C01831=1180.589,-28.436,-43.690,179.742,5.773,149.102
C01832=1180.584,-28.186,-43.703,179.744,5.773,149.101
C01833=1180.579,-27.936,-43.716,179.746,5.773,149.101
C01834=1180.573,-27.686,-43.728,179.749,5.774,149.100
C01835=1180.568,-27.437,-43.740,179.751,5.774,149.100
C01836=1180.563,-27.188,-43.753,179.753,5.775,149.099
C01837=1180.557,-26.938,-43.766,179.756,5.775,149.098
C01838=1180.553,-26.687,-43.778,179.758,5.776,149.098
C01839=1180.547,-26.438,-43.791,179.761,5.777,149.097
C01840=1180.542,-26.189,-43.803,179.763,5.776,149.096
C01841=1180.537,-25.939,-43.816,179.766,5.777,149.096
C01842=1180.532,-25.689,-43.828,179.768,5.777,149.095
C01843=1180.527,-25.439,-43.841,179.770,5.778,149.094
C01844=1180.522,-25.190,-43.854,179.773,5.778,149.094
C01845=1180.517,-24.941,-43.866,179.775,5.779,149.093
C01846=1180.512,-24.691,-43.878,179.778,5.780,149.093
C01847=1180.506,-24.442,-43.891,179.780,5.779,149.092
C01848=1180.501,-24.191,-43.904,179.782,5.780,149.091
C01849=1180.496,-23.922,-43.917,179.785,5.781,149.091
C01850=1180.491,-23.652,-43.931,179.787,5.781,149.090
C01851=1180.485,-23.382,-43.945,179.790,5.781,149.089
C01852=1180.479,-23.113,-43.958,179.793,5.782,149.089
C01853=1180.474,-22.863,-43.971,179.795,5.782,149.088
C01854=1180.469,-22.613,-43.984,179.798,5.783,149.087
C01855=1180.463,-22.364,-43.997,179.800,5.784,149.087
C01856=1180.458,-22.115,-44.009,179.803,5.784,149.086
C01857=1180.453,-21.865,-44.022,179.806,5.785,149.085
C01858=1180.449,-21.615,-44.035,179.808,5.785,149.085
C01859=1180.443,-21.365,-44.047,179.810,5.785,149.084
C01860=1180.437,-21.116,-44.060,179.813,5.785,149.084
C01861=1180.433,-20.866,-44.073,179.815,5.786,149.083
C01862=1180.428,-20.616,-44.086,179.817,5.787,149.082
C01863=1180.423,-20.367,-44.098,179.820,5.787,149.082
C01864=1180.417,-20.118,-44.111,179.822,5.788,149.081
C01865=1180.412,-19.867,-44.124,179.825,5.788,149.080
C01866=1180.407,-19.618,-44.137,179.828,5.789,149.080
C01867=1180.402,-19.369,-44.150,179.830,5.789,149.079
C01868=1180.397,-19.119,-44.162,179.832,5.789,149.079
C01869=1180.392,-18.869,-44.176,179.834,5.790,149.078
C01870=1180.386,-18.620,-44.188,179.837,5.790,149.077
C01871=1180.381,-18.370,-44.201,179.839,5.791,149.077
C01872=1180.377,-18.120,-44.214,179.842,5.792,149.076
C01873=1180.371,-17.871,-44.227,179.845,5.792,149.075
C01874=1180.366,-17.621,-44.240,179.847,5.793,149.075
C01875=1180.361,-17.371,-44.253,179.849,5.793,149.074
C01876=1180.355,-17.122,-44.266,179.852,5.794,149.074
C01877=1180.350,-16.872,-44.278,179.854,5.794,149.073
C01878=1180.346,-16.622,-44.291,179.856,5.794,149.072
C01879=1180.341,-16.373,-44.304,179.859,5.795,149.072
C01880=1180.335,-16.124,-44.317,179.862,5.795,149.071
C01881=1180.330,-15.873,-44.330,179.864,5.796,149.071
C01882=1180.325,-15.624,-44.343,179.866,5.796,149.070
C01883=1180.319,-15.375,-44.356,179.869,5.797,149.069
C01884=1180.315,-15.125,-44.369,179.871,5.798,149.069
C01885=1180.310,-14.875,-44.382,179.874,5.798,149.068
C01886=1180.304,-14.626,-44.395,179.877,5.799,149.067
C01887=1180.300,-14.376,-44.408,179.878,5.799,149.067
C01888=1180.294,-14.127,-44.421,179.881,5.799,149.066
C01889=1180.289,-13.877,-44.434,179.884,5.800,149.065
C01890=1180.284,-13.627,-44.447,179.886,5.800,149.065
C01891=1180.278,-13.378,-44.460,179.888,5.801,149.064
C01892=1180.273,-13.128,-44.473,179.891,5.801,149.064
C01893=1180.269,-12.878,-44.486,179.894,5.802,149.063
C01894=1180.263,-12.629,-44.500,179.896,5.803,149.062
C01895=1180.258,-12.379,-44.513,179.899,5.803,149.062
C01896=1180.253,-12.130,-44.525,179.901,5.804,149.061
C01897=1180.247,-11.880,-44.539,179.903,5.804,149.061
C01898=1180.243,-11.630,-44.552,179.906,5.805,149.060
C01899=1180.237,-11.381,-44.566,179.909,5.805,149.059
C01900=1180.233,-11.131,-44.579,179.910,5.805,149.059
C01901=1180.227,-10.882,-44.592,179.913,5.806,149.058
C01902=1180.222,-10.632,-44.605,179.916,5.806,149.057
C01903=1180.218,-10.383,-44.618,179.918,5.807,149.057
C01904=1180.212,-10.133,-44.631,179.920,5.808,149.056
C01905=1180.207,-9.883,-44.644,179.923,5.808,149.055
C01906=1180.201,-9.634,-44.657,179.926,5.809,149.055
C01907=1180.197,-9.384,-44.671,179.928,5.809,149.054
C01908=1180.191,-9.135,-44.684,179.931,5.810,149.054
C01909=1180.187,-8.885,-44.697,179.933,5.810,149.053
C01910=1180.181,-8.635,-44.710,179.935,5.811,149.052
C01911=1180.177,-8.386,-44.724,179.938,5.812,149.052
C01912=1180.171,-8.136,-44.737,179.941,5.812,149.051
C01913=1180.166,-7.887,-44.750,179.943,5.813,149.050
C01914=1180.161,-7.637,-44.764,179.945,5.813,149.050
C01915=1180.156,-7.388,-44.777,179.948,5.814,149.049
C01916=1180.150,-7.137,-44.790,179.950,5.813,149.049
C01917=1180.146,-6.889,-44.804,179.952,5.814,149.048
C01918=1180.140,-6.638,-44.817,179.955,5.815,149.047
C01919=1180.136,-6.390,-44.830,179.958,5.815,149.047
C01920=1180.130,-6.139,-44.844,179.960,5.816,149.046
C01921=1180.125,-5.890,-44.857,179.963,5.817,149.046
C01922=1180.120,-5.640,-44.871,179.965,5.817,149.045
C01923=1180.115,-5.391,-44.884,179.967,5.818,149.044
C01924=1180.110,-5.141,-44.898,179.970,5.818,149.044
C01925=1180.105,-4.892,-44.910,179.973,5.819,149.043
C01926=1180.100,-4.641,-44.924,179.975,5.819,149.042
C01927=1180.094,-4.392,-44.938,179.977,5.820,149.042
C01928=1180.090,-4.142,-44.951,179.980,5.821,149.041
C01929=1180.084,-3.893,-44.965,179.983,5.821,149.040
C01930=1180.080,-3.643,-44.978,179.985,5.822,149.040
C01931=1180.074,-3.394,-44.992,179.988,5.822,149.039
C01932=1180.069,-3.144,-45.005,179.990,5.823,149.039
C01933=1180.064,-2.895,-45.019,179.992,5.824,149.038
C01934=1180.059,-2.645,-45.032,179.995,5.824,149.037
C01935=1180.054,-2.396,-45.046,179.998,5.825,149.037
C01936=1180.049,-2.146,-45.059,180.000,5.825,149.036
C01937=1180.044,-1.896,-45.073,-179.997,5.826,149.036
C01938=1180.039,-1.647,-45.086,-179.995,5.826,149.035
C01939=1180.034,-1.397,-45.100,-179.993,5.827,149.035
C01940=1180.028,-1.148,-45.113,-179.990,5.828,149.034
C01941=1180.023,-0.898,-45.127,-179.987,5.828,149.033
C01942=1180.018,-0.649,-45.140,-179.985,5.829,149.032
C01943=1180.013,-0.399,-45.154,-179.982,5.829,149.032
C01944=1180.008,-0.150,-45.168,-179.980,5.830,149.031
C01945=1180.003,0.100,-45.181,-179.977,5.830,149.031
C01946=1179.998,0.350,-45.196,-179.976,5.830,149.030
C01947=1179.993,0.599,-45.208,-179.973,5.831,149.029
C01948=1179.988,0.849,-45.222,-179.970,5.831,149.029
C01949=1179.983,1.099,-45.237,-179.968,5.832,149.028
C01950=1179.977,1.348,-45.249,-179.965,5.833,149.028
C01951=1179.973,1.598,-45.264,-179.963,5.833,149.027
C01952=1179.967,1.847,-45.277,-179.961,5.834,149.026
C01953=1179.961,2.117,-45.292,-179.957,5.835,149.026
C01954=1179.956,2.386,-45.307,-179.955,5.836,149.025
C01955=1179.951,2.655,-45.321,-179.952,5.836,149.024
C01956=1179.945,2.924,-45.336,-179.949,5.837,149.024
C01957=1179.940,3.174,-45.350,-179.947,5.837,149.023
C01958=1179.935,3.423,-45.364,-179.945,5.838,149.023
C01959=1179.929,3.673,-45.378,-179.942,5.838,149.022
C01960=1179.925,3.922,-45.391,-179.939,5.839,149.021
C01961=1179.920,4.172,-45.406,-179.937,5.840,149.021
C01962=1179.915,4.421,-45.419,-179.934,5.840,149.020
C01963=1179.909,4.671,-45.433,-179.932,5.841,149.019
C01964=1179.904,4.921,-45.447,-179.930,5.842,149.019
C01965=1179.900,5.170,-45.461,-179.927,5.842,149.018
C01966=1179.895,5.419,-45.475,-179.924,5.843,149.018
C01967=1179.889,5.670,-45.488,-179.922,5.843,149.017
C01968=1179.884,5.919,-45.502,-179.920,5.844,149.016
C01969=1179.879,6.169,-45.517,-179.917,5.844,149.016
C01970=1179.875,6.418,-45.530,-179.914,5.845,149.015
C01971=1179.869,6.667,-45.544,-179.912,5.846,149.015
C01972=1179.864,6.917,-45.558,-179.909,5.846,149.014
C01973=1179.859,7.167,-45.572,-179.907,5.847,149.013
C01974=1179.853,7.416,-45.586,-179.905,5.847,149.013
C01975=1179.848,7.666,-45.600,-179.902,5.848,149.012
C01976=1179.843,7.915,-45.615,-179.899,5.848,149.011
C01977=1179.839,8.165,-45.628,-179.897,5.849,149.011
C01978=1179.833,8.414,-45.641,-179.894,5.850,149.010
C01979=1179.828,8.664,-45.656,-179.892,5.850,149.010
C01980=1179.823,8.914,-45.670,-179.890,5.851,149.009
C01981=1179.818,9.163,-45.684,-179.887,5.852,149.008
C01982=1179.813,9.413,-45.698,-179.884,5.853,149.008
C01983=1179.808,9.662,-45.712,-179.882,5.854,149.007
C01984=1179.803,9.912,-45.727,-179.879,5.854,149.007
C01985=1179.797,10.161,-45.741,-179.876,5.855,149.006
C01986=1179.793,10.410,-45.754,-179.874,5.855,149.005
C01987=1179.788,10.661,-45.768,-179.871,5.856,149.005
C01988=1179.783,10.910,-45.782,-179.869,5.856,149.004
C01989=1179.777,11.159,-45.796,-179.867,5.857,149.004
C01990=1179.772,11.409,-45.810,-179.864,5.858,149.003
C01991=1179.767,11.659,-45.825,-179.861,5.858,149.002
C01992=1179.763,11.909,-45.839,-179.859,5.859,149.002
C01993=1179.757,12.158,-45.853,-179.857,5.860,149.001
C01994=1179.752,12.407,-45.867,-179.854,5.860,149.000
C01995=1179.747,12.657,-45.881,-179.852,5.861,149.000
C01996=1179.742,12.907,-45.896,-179.849,5.861,148.999
C01997=1179.737,13.156,-45.910,-179.846,5.862,148.999
C01998=1179.732,13.405,-45.924,-179.844,5.863,148.998
C01999=1179.727,13.655,-45.938,-179.842,5.863,148.997
C02000=1179.722,13.905,-45.952,-179.839,5.864,148.997
C02001=1179.717,14.155,-45.967,-179.837,5.865,148.996
C02002=1179.711,14.403,-45.981,-179.834,5.865,148.996
C02003=1179.707,14.653,-45.996,-179.831,5.866,148.995
C02004=1179.702,14.902,-46.010,-179.829,5.867,148.994
C02005=1179.697,15.152,-46.024,-179.826,5.868,148.994
C02006=1179.692,15.402,-46.038,-179.823,5.868,148.993
C02007=1179.687,15.652,-46.053,-179.821,5.869,148.993
C02008=1179.681,15.901,-46.067,-179.819,5.869,148.992
C02009=1179.676,16.150,-46.081,-179.816,5.870,148.991
C02010=1179.671,16.400,-46.095,-179.814,5.871,148.991
C02011=1179.666,16.650,-46.109,-179.811,5.871,148.990
C02012=1179.661,16.899,-46.125,-179.808,5.872,148.989
C02013=1179.656,17.149,-46.139,-179.806,5.873,148.989
C02014=1179.650,17.398,-46.153,-179.804,5.873,148.988
C02015=1179.645,17.648,-46.167,-179.801,5.874,148.988
C02016=1179.640,17.897,-46.182,-179.799,5.874,148.987
C02017=1179.636,18.147,-46.196,-179.796,5.876,148.986
C02018=1179.631,18.396,-46.211,-179.793,5.876,148.986
C02019=1179.626,18.646,-46.225,-179.791,5.877,148.985
C02020=1179.621,18.895,-46.240,-179.788,5.878,148.985
C02021=1179.616,19.145,-46.254,-179.786,5.878,148.984
C02022=1179.610,19.394,-46.269,-179.783,5.879,148.984
C02023=1179.605,19.644,-46.283,-179.781,5.879,148.983
C02024=1179.600,19.893,-46.298,-179.778,5.880,148.982
C02025=1179.595,20.143,-46.312,-179.776,5.881,148.982
C02026=1179.591,20.392,-46.327,-179.773,5.881,148.981
C02027=1179.586,20.642,-46.341,-179.771,5.882,148.980
C02028=1179.580,20.892,-46.356,-179.768,5.883,148.980
C02029=1179.575,21.142,-46.370,-179.765,5.884,148.979
C02030=1179.570,21.391,-46.385,-179.763,5.884,148.979
C02031=1179.565,21.640,-46.400,-179.760,5.885,148.978
C02032=1179.560,21.890,-46.414,-179.758,5.886,148.977
C02033=1179.554,22.139,-46.429,-179.755,5.886,148.977
C02034=1179.549,22.388,-46.443,-179.753,5.887,148.976
C02035=1179.544,22.638,-46.458,-179.750,5.887,148.976
C02036=1179.540,22.887,-46.473,-179.748,5.888,148.975
C02037=1179.535,23.137,-46.487,-179.745,5.889,148.974
C02038=1179.529,23.387,-46.502,-179.742,5.890,148.974
C02039=1179.525,23.636,-46.517,-179.740,5.891,148.973
C02040=1179.520,23.886,-46.531,-179.737,5.891,148.973
C02041=1179.515,24.135,-46.546,-179.735,5.892,148.972
C02042=1179.509,24.385,-46.561,-179.732,5.892,148.971
C02043=1179.504,24.635,-46.575,-179.730,5.893,148.971
C02044=1179.500,24.884,-46.590,-179.727,5.894,148.970
C02045=1179.495,25.133,-46.604,-179.725,5.895,148.970
C02046=1179.489,25.383,-46.620,-179.722,5.896,148.969
C02047=1179.484,25.633,-46.634,-179.719,5.896,148.968
C02048=1179.480,25.882,-46.649,-179.717,5.897,148.968
C02049=1179.474,26.132,-46.664,-179.714,5.898,148.967
C02050=1179.469,26.381,-46.679,-179.712,5.898,148.967
C02051=1179.464,26.630,-46.693,-179.710,5.899,148.966
C02052=1179.459,26.880,-46.709,-179.707,5.900,148.965
C02053=1179.454,27.130,-46.723,-179.704,5.900,148.965
C02054=1179.449,27.379,-46.738,-179.702,5.902,148.964
C02055=1179.444,27.629,-46.753,-179.699,5.902,148.964
C02056=1179.439,27.878,-46.768,-179.696,5.903,148.963
C02057=1179.434,28.147,-46.784,-179.694,5.904,148.962
C02058=1179.428,28.416,-46.800,-179.692,5.904,148.962
C02059=1179.423,28.684,-46.816,-179.688,5.905,148.961
C02060=1179.417,28.954,-46.832,-179.686,5.906,148.960
C02061=1179.412,29.203,-46.847,-179.683,5.906,148.960
C02062=1179.407,29.452,-46.861,-179.681,5.907,148.959
C02063=1179.402,29.702,-46.877,-179.678,5.908,148.959
C02064=1179.397,29.951,-46.891,-179.675,5.909,148.958
C02065=1179.392,30.201,-46.907,-179.673,5.910,148.957
C02066=1179.387,30.450,-46.922,-179.670,5.910,148.957
C02067=1179.382,30.700,-46.936,-179.668,5.911,148.956
C02068=1179.377,30.949,-46.952,-179.665,5.912,148.956
C02069=1179.372,31.198,-46.967,-179.663,5.912,148.955
C02070=1179.366,31.448,-46.982,-179.660,5.914,148.955
C02071=1179.362,31.698,-46.997,-179.657,5.914,148.954
C02072=1179.357,31.947,-47.013,-179.655,5.915,148.953
C02073=1179.352,32.197,-47.027,-179.653,5.916,148.953
C02074=1179.347,32.446,-47.042,-179.650,5.916,148.952
C02075=1179.342,32.696,-47.057,-179.647,5.917,148.951
C02076=1179.337,32.945,-47.072,-179.644,5.918,148.951
C02077=1179.332,33.195,-47.087,-179.642,5.919,148.950
C02078=1179.327,33.444,-47.102,-179.640,5.920,148.950
C02079=1179.321,33.694,-47.117,-179.637,5.920,148.949
C02080=1179.317,33.943,-47.132,-179.634,5.921,148.948
C02081=1179.312,34.193,-47.148,-179.632,5.922,148.948
C02082=1179.307,34.442,-47.163,-179.629,5.923,148.947
C02083=1179.302,34.692,-47.178,-179.626,5.923,148.947
C02084=1179.297,34.941,-47.193,-179.624,5.924,148.946
C02085=1179.291,35.191,-47.209,-179.622,5.925,148.946
C02086=1179.287,35.440,-47.224,-179.619,5.926,148.945
C02087=1179.281,35.689,-47.239,-179.617,5.926,148.944
C02088=1179.277,35.940,-47.254,-179.614,5.928,148.944
C02089=1179.272,36.189,-47.269,-179.611,5.928,148.943
C02090=1179.266,36.438,-47.285,-179.609,5.929,148.943
C02091=1179.262,36.687,-47.300,-179.606,5.929,148.942
C02092=1179.256,36.937,-47.316,-179.604,5.930,148.942
C02093=1179.252,37.186,-47.331,-179.601,5.932,148.941
C02094=1179.247,37.437,-47.346,-179.599,5.932,148.940
C02095=1179.242,37.686,-47.361,-179.596,5.933,148.940
C02096=1179.236,37.935,-47.376,-179.593,5.933,148.939
C02097=1179.231,38.185,-47.392,-179.591,5.934,148.939
C02098=1179.226,38.434,-47.407,-179.588,5.936,148.938
C02099=1179.221,38.683,-47.423,-179.586,5.936,148.937
C02100=1179.217,38.933,-47.438,-179.583,5.937,148.937
C02101=1179.212,39.182,-47.453,-179.580,5.937,148.936
C02102=1179.206,39.432,-47.469,-179.578,5.938,148.936
C02103=1179.202,39.681,-47.484,-179.575,5.940,148.935
C02104=1179.196,39.930,-47.500,-179.572,5.940,148.934
C02105=1179.191,40.181,-47.515,-179.570,5.941,148.934
C02106=1179.186,40.430,-47.530,-179.568,5.942,148.933
C02107=1179.181,40.679,-47.545,-179.565,5.942,148.933
C02108=1179.176,40.929,-47.561,-179.562,5.944,148.932
C02109=1179.172,41.179,-47.576,-179.560,5.944,148.931
C02110=1179.166,41.428,-47.592,-179.557,5.945,148.931
C02111=1179.161,41.677,-47.608,-179.555,5.946,148.930
C02112=1179.156,41.926,-47.623,-179.553,5.946,148.930
C02113=1179.151,42.177,-47.639,-179.549,5.948,148.929
C02114=1179.146,42.426,-47.654,-179.547,5.948,148.929
C02115=1179.142,42.674,-47.670,-179.545,5.949,148.928
C02116=1179.136,42.924,-47.685,-179.542,5.950,148.927
C02117=1179.132,43.174,-47.701,-179.539,5.951,148.927
C02118=1179.126,43.423,-47.717,-179.537,5.952,148.926
C02119=1179.122,43.672,-47.732,-179.534,5.952,148.926
C02120=1179.116,43.922,-47.748,-179.532,5.953,148.925
C02121=1179.111,44.172,-47.764,-179.529,5.954,148.925
C02122=1179.106,44.421,-47.779,-179.526,5.955,148.924
C02123=1179.101,44.670,-47.794,-179.524,5.956,148.923
C02124=1179.097,44.920,-47.810,-179.521,5.956,148.923
C02125=1179.091,45.169,-47.826,-179.519,5.957,148.922
C02126=1179.086,45.419,-47.842,-179.516,5.959,148.922
C02127=1179.082,45.668,-47.857,-179.514,5.959,148.921
C02128=1179.077,45.918,-47.873,-179.511,5.960,148.921
C02129=1179.071,46.167,-47.888,-179.508,5.960,148.920
C02130=1179.066,46.417,-47.904,-179.506,5.962,148.919
C02131=1179.061,46.666,-47.921,-179.503,5.963,148.919
C02132=1179.057,46.915,-47.936,-179.501,5.964,148.918
C02133=1179.052,47.165,-47.952,-179.498,5.964,148.918
C02134=1179.047,47.415,-47.967,-179.495,5.965,148.917
C02135=1179.041,47.664,-47.983,-179.493,5.966,148.917
C02136=1179.037,47.914,-48.000,-179.490,5.967,148.916
C02137=1179.031,48.163,-48.015,-179.488,5.968,148.915
C02138=1179.027,48.412,-48.030,-179.485,5.969,148.915
C02139=1179.022,48.662,-48.046,-179.482,5.969,148.914
C02140=1179.017,48.911,-48.062,-179.480,5.970,148.914
C02141=1179.011,49.160,-48.078,-179.477,5.971,148.913
C02142=1179.007,49.411,-48.094,-179.475,5.973,148.913
C02143=1179.002,49.659,-48.110,-179.472,5.973,148.912
C02144=1178.997,49.909,-48.126,-179.469,5.974,148.911
C02145=1178.991,50.159,-48.142,-179.467,5.974,148.911
C02146=1178.987,50.407,-48.157,-179.464,5.976,148.910
C02147=1178.982,50.657,-48.173,-179.462,5.977,148.910
C02148=1178.977,50.907,-48.189,-179.459,5.977,148.909
C02149=1178.972,51.156,-48.206,-179.457,5.978,148.909
C02150=1178.967,51.406,-48.221,-179.454,5.979,148.908
C02151=1178.962,51.655,-48.237,-179.451,5.980,148.907
C02152=1178.957,51.905,-48.254,-179.449,5.981,148.907
C02153=1178.952,52.154,-48.269,-179.446,5.982,148.906
C02154=1178.947,52.404,-48.285,-179.444,5.983,148.906
C02155=1178.942,52.653,-48.301,-179.441,5.983,148.905
C02156=1178.937,52.903,-48.317,-179.439,5.984,148.905
C02157=1178.932,53.152,-48.334,-179.436,5.986,148.904
C02158=1178.927,53.401,-48.349,-179.433,5.986,148.903
C02159=1178.922,53.651,-48.366,-179.431,5.987,148.903
C02160=1178.917,53.900,-48.381,-179.428,5.988,148.902
C02161=1178.912,54.169,-48.399,-179.425,5.989,148.901
C02162=1178.907,54.437,-48.417,-179.423,5.990,148.901
C02163=1178.901,54.706,-48.434,-179.420,5.991,148.900
C02164=1178.895,54.974,-48.451,-179.417,5.992,148.900
C02165=1178.891,55.224,-48.467,-179.414,5.993,148.899
C02166=1178.886,55.473,-48.483,-179.412,5.994,148.899
C02167=1178.881,55.722,-48.500,-179.409,5.994,148.898
C02168=1178.876,55.972,-48.515,-179.406,5.996,148.897
C02169=1178.871,56.221,-48.532,-179.404,5.996,148.897
C02170=1178.866,56.471,-48.547,-179.401,5.997,148.896
C02171=1178.861,56.720,-48.564,-179.398,5.999,148.896
C02172=1178.856,56.970,-48.580,-179.396,6.000,148.895
C02173=1178.851,57.219,-48.597,-179.393,6.000,148.895
C02174=1178.845,57.469,-48.612,-179.391,6.001,148.894
C02175=1178.841,57.718,-48.629,-179.388,6.002,148.893
C02176=1178.836,57.967,-48.645,-179.385,6.003,148.893
C02177=1178.831,58.217,-48.661,-179.383,6.004,148.892
C02178=1178.826,58.466,-48.678,-179.380,6.005,148.892
C02179=1178.821,58.715,-48.694,-179.378,6.006,148.891
C02180=1178.816,58.965,-48.710,-179.375,6.006,148.891
C02181=1178.812,59.214,-48.727,-179.373,6.008,148.890
C02182=1178.805,59.464,-48.743,-179.370,6.009,148.889
C02183=1178.801,59.713,-48.759,-179.368,6.010,148.889
C02184=1178.796,59.963,-48.776,-179.365,6.011,148.888
C02185=1178.791,60.212,-48.792,-179.362,6.011,148.888
C02186=1178.787,60.462,-48.808,-179.360,6.012,148.887
C02187=1178.782,60.711,-48.825,-179.357,6.014,148.887
C02188=1178.777,60.960,-48.841,-179.354,6.014,148.886
C02189=1178.771,61.210,-48.858,-179.352,6.015,148.886
C02190=1178.766,61.459,-48.874,-179.349,6.017,148.885
C02191=1178.762,61.709,-48.891,-179.346,6.017,148.884
C02192=1178.757,61.958,-48.907,-179.344,6.018,148.884
C02193=1178.752,62.208,-48.923,-179.341,6.019,148.883
C02194=1178.746,62.457,-48.940,-179.339,6.020,148.883
C02195=1178.742,62.706,-48.957,-179.336,6.021,148.882
C02196=1178.737,62.955,-48.973,-179.333,6.022,148.882
C02197=1178.732,63.205,-48.989,-179.331,6.023,148.881
C02198=1178.727,63.455,-49.006,-179.328,6.024,148.880
C02199=1178.722,63.704,-49.023,-179.325,6.025,148.880
C02200=1178.717,63.953,-49.039,-179.323,6.026,148.879
C02201=1178.713,64.203,-49.056,-179.321,6.027,148.879
C02202=1178.707,64.452,-49.073,-179.317,6.028,148.878
C02203=1178.702,64.702,-49.089,-179.315,6.029,148.878
C02204=1178.697,64.951,-49.105,-179.313,6.029,148.877
C02205=1178.692,65.200,-49.122,-179.310,6.031,148.877
C02206=1178.687,65.450,-49.139,-179.307,6.032,148.876
C02207=1178.682,65.699,-49.155,-179.305,6.033,148.876
C02208=1178.678,65.948,-49.172,-179.302,6.034,148.875
C02209=1178.672,66.198,-49.189,-179.300,6.035,148.875
C02210=1178.667,66.447,-49.206,-179.297,6.036,148.874
C02211=1178.663,66.696,-49.222,-179.294,6.037,148.873
C02212=1178.658,66.946,-49.239,-179.292,6.037,148.873
C02213=1178.653,67.195,-49.256,-179.289,6.039,148.872
C02214=1178.648,67.444,-49.272,-179.286,6.040,148.872
C02215=1178.643,67.695,-49.289,-179.284,6.040,148.871
C02216=1178.638,67.944,-49.305,-179.281,6.042,148.871
C02217=1178.633,68.193,-49.322,-179.278,6.042,148.870
C02218=1178.628,68.443,-49.339,-179.276,6.044,148.870
C02219=1178.623,68.692,-49.356,-179.273,6.045,148.869
C02220=1178.618,68.941,-49.372,-179.271,6.046,148.868
C02221=1178.613,69.191,-49.389,-179.268,6.047,148.868
C02222=1178.609,69.440,-49.407,-179.266,6.048,148.867
C02223=1178.603,69.689,-49.424,-179.263,6.048,148.867
C02224=1178.599,69.938,-49.440,-179.260,6.050,148.866
C02225=1178.594,70.188,-49.457,-179.258,6.051,148.866
C02226=1178.589,70.438,-49.474,-179.255,6.052,148.865
C02227=1178.584,70.686,-49.491,-179.252,6.053,148.865
C02228=1178.579,70.936,-49.508,-179.250,6.054,148.864
C02229=1178.574,71.186,-49.525,-179.247,6.055,148.863
C02230=1178.569,71.435,-49.542,-179.245,6.056,148.863
C02231=1178.564,71.684,-49.558,-179.242,6.057,148.862
C02232=1178.559,71.934,-49.575,-179.239,6.058,148.862
C02233=1178.554,72.184,-49.592,-179.237,6.059,148.861
C02234=1178.550,72.432,-49.609,-179.234,6.060,148.861
C02235=1178.544,72.681,-49.626,-179.231,6.061,148.860
C02236=1178.540,72.931,-49.643,-179.229,6.063,148.860
C02237=1178.534,73.181,-49.660,-179.226,6.063,148.859
C02238=1178.530,73.430,-49.677,-179.224,6.064,148.859
C02239=1178.524,73.679,-49.695,-179.221,6.065,148.858
C02240=1178.520,73.928,-49.711,-179.219,6.066,148.858
C02241=1178.515,74.178,-49.729,-179.215,6.068,148.857
C02242=1178.510,74.427,-49.745,-179.213,6.068,148.856
C02243=1178.505,74.677,-49.762,-179.210,6.070,148.856
C02244=1178.500,74.925,-49.779,-179.208,6.071,148.855
C02245=1178.495,75.175,-49.797,-179.205,6.071,148.855
C02246=1178.490,75.425,-49.814,-179.203,6.073,148.854
C02247=1178.485,75.675,-49.831,-179.200,6.073,148.854
C02248=1178.480,75.924,-49.849,-179.197,6.075,148.853
C02249=1178.476,76.173,-49.865,-179.195,6.076,148.853
C02250=1178.470,76.422,-49.882,-179.192,6.077,148.852
C02251=1178.466,76.671,-49.900,-179.189,6.078,148.852
C02252=1178.461,76.921,-49.917,-179.187,6.079,148.851
C02253=1178.456,77.171,-49.934,-179.184,6.080,148.850
C02254=1178.451,77.420,-49.952,-179.182,6.081,148.850
C02255=1178.446,77.669,-49.969,-179.178,6.082,148.849
C02256=1178.441,77.918,-49.985,-179.176,6.083,148.849
C02257=1178.436,78.167,-50.003,-179.173,6.085,148.848
C02258=1178.431,78.417,-50.020,-179.171,6.086,148.848
C02259=1178.426,78.667,-50.037,-179.168,6.086,148.847
C02260=1178.422,78.916,-50.055,-179.166,6.088,148.847
C02261=1178.416,79.166,-50.072,-179.163,6.088,148.846
C02262=1178.412,79.414,-50.090,-179.160,6.090,148.846
C02263=1178.407,79.664,-50.107,-179.158,6.091,148.845
C02264=1178.401,79.913,-50.124,-179.155,6.092,148.845
C02265=1178.397,80.181,-50.143,-179.152,6.093,148.844
C02266=1178.391,80.450,-50.161,-179.150,6.094,148.844
C02267=1178.386,80.719,-50.180,-179.146,6.096,148.843
C02268=1178.380,80.987,-50.199,-179.144,6.096,148.842
C02269=1178.376,81.236,-50.216,-179.141,6.098,148.842
C02270=1178.371,81.485,-50.234,-179.138,6.099,148.841
C02271=1178.366,81.735,-50.251,-179.136,6.100,148.841
C02272=1178.361,81.984,-50.269,-179.134,6.101,148.840
C02273=1178.356,82.234,-50.286,-179.131,6.102,148.840
C02274=1178.351,82.483,-50.304,-179.128,6.103,148.839
C02275=1178.346,82.733,-50.321,-179.126,6.104,148.839
C02276=1178.341,82.982,-50.339,-179.123,6.106,148.838
C02277=1178.337,83.231,-50.355,-179.120,6.106,148.837
C02278=1178.332,83.481,-50.373,-179.117,6.108,148.837
C02279=1178.327,83.730,-50.391,-179.115,6.108,148.836
C02280=1178.322,83.979,-50.409,-179.112,6.110,148.836
C02281=1178.318,84.228,-50.426,-179.109,6.111,148.835
C02282=1178.312,84.478,-50.443,-179.107,6.112,148.835
C02283=1178.307,84.727,-50.461,-179.104,6.113,148.834
C02284=1178.303,84.977,-50.479,-179.101,6.115,148.834
C02285=1178.297,85.226,-50.496,-179.099,6.116,148.833
C02286=1178.293,85.474,-50.514,-179.096,6.117,148.833
C02287=1178.288,85.724,-50.532,-179.094,6.118,148.832
C02288=1178.282,85.973,-50.549,-179.091,6.119,148.832
C02289=1178.277,86.223,-50.567,-179.089,6.120,148.831
C02290=1178.273,86.472,-50.585,-179.085,6.121,148.831
C02291=1178.268,86.722,-50.602,-179.083,6.122,148.830
C02292=1178.264,86.971,-50.620,-179.080,6.124,148.830
C02293=1178.259,87.220,-50.638,-179.078,6.125,148.829
C02294=1178.254,87.470,-50.655,-179.075,6.126,148.829
C02295=1178.249,87.719,-50.673,-179.073,6.127,148.828
C02296=1178.244,87.968,-50.691,-179.070,6.129,148.828
C02297=1178.239,88.218,-50.709,-179.067,6.129,148.827
C02298=1178.234,88.467,-50.726,-179.064,6.131,148.827
C02299=1178.229,88.717,-50.744,-179.062,6.131,148.826
C02300=1178.224,88.966,-50.762,-179.059,6.133,148.826
C02301=1178.220,89.215,-50.780,-179.057,6.134,148.825
C02302=1178.215,89.464,-50.798,-179.054,6.135,148.824
C02303=1178.210,89.714,-50.815,-179.052,6.136,148.824
C02304=1178.205,89.963,-50.833,-179.048,6.138,148.823
C02305=1178.200,90.212,-50.851,-179.046,6.138,148.823
C02306=1178.195,90.461,-50.869,-179.043,6.140,148.822
C02307=1178.190,90.710,-50.887,-179.041,6.141,148.822
C02308=1178.185,90.959,-50.905,-179.038,6.142,148.821
C02309=1178.180,91.209,-50.922,-179.036,6.143,148.821
C02310=1178.175,91.459,-50.940,-179.033,6.145,148.820
C02311=1178.171,91.708,-50.958,-179.030,6.145,148.820
C02312=1178.166,91.958,-50.976,-179.028,6.147,148.819
C02313=1178.161,92.207,-50.994,-179.025,6.148,148.819
C02314=1178.156,92.456,-51.012,-179.022,6.149,148.818
C02315=1178.151,92.705,-51.030,-179.020,6.150,148.818
C02316=1178.146,92.954,-51.048,-179.017,6.151,148.817
C02317=1178.141,93.203,-51.066,-179.015,6.152,148.817
C02318=1178.136,93.453,-51.084,-179.012,6.154,148.816
C02319=1178.132,93.702,-51.103,-179.009,6.155,148.816
C02320=1178.127,93.952,-51.121,-179.007,6.156,148.815
C02321=1178.122,94.201,-51.139,-179.004,6.158,148.815
C02322=1178.117,94.450,-51.156,-179.001,6.159,148.814
C02323=1178.112,94.699,-51.174,-178.998,6.160,148.814
C02324=1178.107,94.948,-51.192,-178.996,6.161,148.813
C02325=1178.102,95.198,-51.211,-178.993,6.163,148.813
C02326=1178.097,95.448,-51.229,-178.991,6.163,148.812
C02327=1178.092,95.697,-51.247,-178.988,6.165,148.812
C02328=1178.088,95.946,-51.265,-178.985,6.165,148.811
C02329=1178.083,96.195,-51.283,-178.983,6.167,148.811
C02330=1178.078,96.444,-51.301,-178.980,6.169,148.810
C02331=1178.073,96.694,-51.320,-178.977,6.169,148.810
C02332=1178.068,96.943,-51.338,-178.975,6.171,148.809
C02333=1178.064,97.193,-51.356,-178.972,6.172,148.809
C02334=1178.058,97.442,-51.374,-178.969,6.173,148.808
C02335=1178.053,97.691,-51.393,-178.967,6.174,148.808
C02336=1178.048,97.940,-51.411,-178.964,6.176,148.807
C02337=1178.044,98.190,-51.429,-178.961,6.177,148.807
C02338=1178.039,98.439,-51.447,-178.959,6.178,148.806
C02339=1178.034,98.688,-51.465,-178.956,6.180,148.806
C02340=1178.029,98.938,-51.484,-178.954,6.181,148.805
C02341=1178.025,99.187,-51.503,-178.951,6.182,148.805
C02342=1178.020,99.436,-51.521,-178.948,6.183,148.804
C02343=1178.015,99.685,-51.539,-178.946,6.185,148.804
C02344=1178.010,99.934,-51.557,-178.942,6.186,148.803
C02345=1178.005,100.185,-51.576,-178.940,6.187,148.803
C02346=1178.000,100.433,-51.594,-178.937,6.188,148.802
C02347=1177.995,100.682,-51.612,-178.935,6.189,148.802
C02348=1177.990,100.931,-51.630,-178.932,6.191,148.801
C02349=1177.985,101.182,-51.649,-178.930,6.191,148.801
C02350=1177.981,101.430,-51.668,-178.927,6.193,148.800
C02351=1177.976,101.679,-51.686,-178.924,6.195,148.800
C02352=1177.971,101.929,-51.704,-178.922,6.195,148.799
C02353=1177.966,102.178,-51.724,-178.919,6.197,148.799
C02354=1177.961,102.427,-51.742,-178.917,6.198,148.798
C02355=1177.956,102.676,-51.760,-178.914,6.199,148.798
C02356=1177.951,102.927,-51.778,-178.911,6.201,148.797
C02357=1177.947,103.175,-51.797,-178.908,6.202,148.797
C02358=1177.942,103.424,-51.815,-178.906,6.203,148.796
C02359=1177.937,103.673,-51.834,-178.903,6.204,148.796
C02360=1177.932,103.923,-51.853,-178.900,6.206,148.795
C02361=1177.927,104.172,-51.871,-178.898,6.207,148.795
C02362=1177.923,104.421,-51.889,-178.895,6.208,148.794
C02363=1177.918,104.671,-51.908,-178.892,6.210,148.794
C02364=1177.913,104.920,-51.927,-178.890,6.211,148.793
C02365=1177.908,105.169,-51.945,-178.887,6.212,148.793
C02366=1177.903,105.419,-51.964,-178.884,6.214,148.792
C02367=1177.898,105.668,-51.983,-178.882,6.215,148.792
C02368=1177.893,105.917,-52.001,-178.879,6.216,148.791
C02369=1177.889,106.185,-52.022,-178.876,6.218,148.791
C02370=1177.883,106.454,-52.042,-178.873,6.219,148.790
C02371=1177.878,106.722,-52.061,-178.871,6.220,148.790
C02372=1177.873,106.991,-52.082,-178.868,6.221,148.789
C02373=1177.868,107.240,-52.100,-178.865,6.223,148.789
C02374=1177.862,107.489,-52.120,-178.863,6.224,148.788
C02375=1177.858,107.739,-52.138,-178.860,6.225,148.788
C02376=1177.853,107.988,-52.157,-178.857,6.227,148.787
C02377=1177.849,108.237,-52.176,-178.855,6.228,148.787
C02378=1177.844,108.486,-52.194,-178.852,6.229,148.786
C02379=1177.839,108.735,-52.214,-178.849,6.231,148.786
C02380=1177.834,108.985,-52.232,-178.847,6.232,148.785
C02381=1177.829,109.234,-52.251,-178.843,6.233,148.785
C02382=1177.825,109.484,-52.269,-178.841,6.235,148.784
C02383=1177.819,109.732,-52.289,-178.839,6.236,148.784
C02384=1177.815,109.981,-52.307,-178.835,6.237,148.783
C02385=1177.810,110.231,-52.326,-178.833,6.238,148.783
C02386=1177.805,110.480,-52.345,-178.831,6.240,148.782
C02387=1177.800,110.729,-52.365,-178.828,6.242,148.782
C02388=1177.795,110.978,-52.383,-178.825,6.242,148.781
C02389=1177.791,111.228,-52.402,-178.823,6.244,148.781
C02390=1177.786,111.477,-52.421,-178.820,6.246,148.781
C02391=1177.781,111.727,-52.440,-178.817,6.246,148.780
C02392=1177.776,111.975,-52.459,-178.815,6.248,148.779
C02393=1177.771,112.224,-52.478,-178.812,6.250,148.779
C02394=1177.766,112.474,-52.497,-178.809,6.250,148.778
C02395=1177.761,112.723,-52.516,-178.806,6.252,148.778
C02396=1177.757,112.972,-52.535,-178.804,6.254,148.778
C02397=1177.752,113.221,-52.554,-178.801,6.254,148.777
C02398=1177.747,113.471,-52.573,-178.798,6.256,148.777
C02399=1177.742,113.720,-52.592,-178.796,6.258,148.776
C02400=1177.738,113.969,-52.611,-178.793,6.258,148.776
C02401=1177.732,114.218,-52.631,-178.790,6.260,148.775
C02402=1177.728,114.468,-52.649,-178.788,6.262,148.775
C02403=1177.723,114.717,-52.668,-178.786,6.263,148.774
C02404=1177.718,114.967,-52.688,-178.782,6.264,148.774
C02405=1177.713,115.215,-52.707,-178.780,6.266,148.773
C02406=1177.709,115.465,-52.726,-178.778,6.267,148.773
C02407=1177.703,115.714,-52.746,-178.774,6.268,148.772
C02408=1177.699,115.963,-52.765,-178.772,6.270,148.772
C02409=1177.694,116.212,-52.783,-178.769,6.272,148.771
C02410=1177.689,116.462,-52.803,-178.767,6.273,148.771
C02411=1177.684,116.710,-52.822,-178.764,6.274,148.770
C02412=1177.679,116.960,-52.841,-178.761,6.276,148.770
C02413=1177.675,117.210,-52.861,-178.759,6.277,148.770
C02414=1177.670,117.458,-52.880,-178.756,6.278,148.769
C02415=1177.665,117.708,-52.899,-178.753,6.280,148.769
C02416=1177.660,117.957,-52.918,-178.751,6.281,148.768
C02417=1177.656,118.206,-52.938,-178.748,6.282,148.768
C02418=1177.651,118.455,-52.957,-178.745,6.284,148.767
C02419=1177.646,118.704,-52.976,-178.743,6.285,148.767
C02420=1177.641,118.954,-52.996,-178.740,6.286,148.766
C02421=1177.637,119.202,-53.015,-178.737,6.288,148.766
C02422=1177.632,119.452,-53.034,-178.734,6.289,148.765
C02423=1177.626,119.701,-53.054,-178.732,6.290,148.765
C02424=1177.622,119.950,-53.073,-178.729,6.292,148.765
C02425=1177.618,120.200,-53.093,-178.726,6.294,148.764
C02426=1177.612,120.448,-53.112,-178.724,6.294,148.763
C02427=1177.608,120.698,-53.131,-178.721,6.296,148.763
C02428=1177.602,120.947,-53.151,-178.719,6.298,148.763
C02429=1177.598,121.196,-53.170,-178.715,6.299,148.762
C02430=1177.594,121.446,-53.189,-178.713,6.300,148.762
C02431=1177.588,121.695,-53.209,-178.711,6.302,148.761
C02432=1177.583,121.944,-53.228,-178.708,6.304,148.761
C02433=1177.579,122.194,-53.248,-178.705,6.305,148.760
C02434=1177.574,122.442,-53.268,-178.703,6.306,148.760
C02435=1177.569,122.692,-53.288,-178.700,6.308,148.759
C02436=1177.565,122.941,-53.307,-178.697,6.309,148.759
C02437=1177.560,123.190,-53.326,-178.695,6.310,148.758
C02438=1177.555,123.439,-53.346,-178.692,6.312,148.758
C02439=1177.550,123.689,-53.365,-178.689,6.314,148.758
C02440=1177.545,123.937,-53.385,-178.686,6.315,148.757
C02441=1177.540,124.187,-53.405,-178.684,6.316,148.757
C02442=1177.536,124.436,-53.425,-178.681,6.318,148.756
C02443=1177.530,124.685,-53.444,-178.678,6.319,148.756
C02444=1177.525,124.935,-53.464,-178.676,6.321,148.755
C02445=1177.522,125.183,-53.483,-178.673,6.322,148.755
C02446=1177.516,125.432,-53.503,-178.670,6.323,148.754
C02447=1177.512,125.682,-53.522,-178.668,6.325,148.754
C02448=1177.507,125.931,-53.543,-178.665,6.327,148.754
C02449=1177.503,126.180,-53.562,-178.662,6.327,148.753
C02450=1177.497,126.429,-53.582,-178.660,6.329,148.753
C02451=1177.492,126.679,-53.601,-178.657,6.331,148.752
C02452=1177.488,126.928,-53.622,-178.654,6.333,148.752
C02453=1177.483,127.176,-53.641,-178.652,6.333,148.751
C02454=1177.478,127.426,-53.661,-178.649,6.335,148.751
C02455=1177.473,127.675,-53.681,-178.646,6.337,148.750
C02456=1177.469,127.925,-53.701,-178.644,6.338,148.750
C02457=1177.464,128.173,-53.721,-178.641,6.339,148.750
C02458=1177.459,128.422,-53.740,-178.638,6.341,148.749
C02459=1177.454,128.672,-53.760,-178.636,6.342,148.749
C02460=1177.450,128.921,-53.780,-178.633,6.344,148.748
C02461=1177.445,129.170,-53.800,-178.630,6.346,148.748
C02462=1177.440,129.419,-53.820,-178.628,6.347,148.747
C02463=1177.435,129.668,-53.840,-178.625,6.348,148.747
C02464=1177.430,129.918,-53.859,-178.622,6.350,148.746
C02465=1177.426,130.167,-53.880,-178.619,6.352,148.746
C02466=1177.421,130.416,-53.899,-178.617,6.353,148.746
C02467=1177.416,130.665,-53.919,-178.614,6.354,148.745
C02468=1177.411,130.914,-53.940,-178.611,6.356,148.745
C02469=1177.406,131.163,-53.960,-178.609,6.358,148.744
C02470=1177.402,131.413,-53.980,-178.606,6.359,148.744
C02471=1177.397,131.661,-54.000,-178.604,6.360,148.743
C02472=1177.392,131.911,-54.019,-178.601,6.362,148.743
C02473=1177.387,132.179,-54.041,-178.598,6.363,148.742
C02474=1177.382,132.448,-54.063,-178.595,6.365,148.742
C02475=1177.377,132.716,-54.084,-178.592,6.367,148.741
C02476=1177.371,132.985,-54.106,-178.589,6.368,148.741
C02477=1177.367,133.234,-54.126,-178.587,6.370,148.741
C02478=1177.362,133.483,-54.146,-178.584,6.372,148.740
C02479=1177.358,133.732,-54.167,-178.581,6.373,148.740
C02480=1177.352,133.982,-54.187,-178.579,6.374,148.739
C02481=1177.348,134.231,-54.207,-178.576,6.376,148.739
C02482=1177.342,134.480,-54.227,-178.573,6.378,148.738
C02483=1177.338,134.729,-54.247,-178.571,6.379,148.738
C02484=1177.334,134.978,-54.267,-178.568,6.381,148.738
C02485=1177.329,135.227,-54.287,-178.565,6.382,148.737
C02486=1177.324,135.477,-54.308,-178.563,6.383,148.737
C02487=1177.319,135.726,-54.328,-178.560,6.385,148.736
C02488=1177.314,135.975,-54.348,-178.557,6.387,148.736
C02489=1177.310,136.224,-54.368,-178.555,6.389,148.735
C02490=1177.305,136.473,-54.389,-178.552,6.390,148.735
C02491=1177.300,136.722,-54.410,-178.549,6.391,148.734
C02492=1177.295,136.971,-54.429,-178.547,6.393,148.734
C02493=1177.291,137.220,-54.449,-178.544,6.394,148.734
C02494=1177.285,137.469,-54.470,-178.541,6.396,148.733
C02495=1177.281,137.718,-54.491,-178.538,6.398,148.733
C02496=1177.276,137.968,-54.510,-178.536,6.400,148.732
C02497=1177.271,138.217,-54.531,-178.533,6.400,148.732
C02498=1177.267,138.466,-54.552,-178.530,6.402,148.731
C02499=1177.262,138.715,-54.572,-178.528,6.404,148.731
C02500=1177.258,138.964,-54.592,-178.525,6.405,148.731
C02501=1177.253,139.213,-54.613,-178.522,6.407,148.730
C02502=1177.248,139.463,-54.633,-178.520,6.409,148.730
C02503=1177.243,139.712,-54.653,-178.517,6.410,148.729
C02504=1177.238,139.961,-54.674,-178.514,6.411,148.729
C02505=1177.234,140.210,-54.695,-178.512,6.413,148.728
C02506=1177.229,140.459,-54.715,-178.509,6.415,148.728
C02507=1177.224,140.708,-54.736,-178.506,6.417,148.728
C02508=1177.220,140.957,-54.757,-178.504,6.418,148.727
C02509=1177.215,141.206,-54.777,-178.501,6.420,148.727
C02510=1177.210,141.455,-54.798,-178.498,6.421,148.726
C02511=1177.206,141.704,-54.818,-178.496,6.422,148.726
C02512=1177.200,141.954,-54.838,-178.493,6.424,148.726
C02513=1177.196,142.203,-54.859,-178.490,6.426,148.725
C02514=1177.191,142.452,-54.880,-178.488,6.428,148.725
C02515=1177.186,142.701,-54.900,-178.485,6.429,148.724
C02516=1177.182,142.950,-54.921,-178.482,6.431,148.724
C02517=1177.177,143.200,-54.942,-178.479,6.433,148.724
C02518=1177.172,143.449,-54.962,-178.477,6.433,148.723
C02519=1177.167,143.698,-54.983,-178.474,6.435,148.723
C02520=1177.163,143.946,-55.004,-178.471,6.437,148.722
C02521=1177.158,144.195,-55.025,-178.469,6.439,148.722
C02522=1177.153,144.444,-55.045,-178.466,6.440,148.721
C02523=1177.148,144.694,-55.066,-178.463,6.442,148.721
C02524=1177.144,144.943,-55.087,-178.461,6.444,148.721
C02525=1177.138,145.192,-55.108,-178.458,6.446,148.720
C02526=1177.134,145.441,-55.128,-178.455,6.446,148.720
C02527=1177.129,145.690,-55.149,-178.453,6.448,148.719
C02528=1177.125,145.940,-55.170,-178.450,6.450,148.719
C02529=1177.120,146.189,-55.191,-178.447,6.452,148.719
C02530=1177.116,146.437,-55.212,-178.445,6.453,148.718
C02531=1177.111,146.687,-55.233,-178.442,6.455,148.718
C02532=1177.106,146.935,-55.253,-178.439,6.457,148.717
C02533=1177.101,147.185,-55.274,-178.437,6.459,148.717
C02534=1177.096,147.434,-55.294,-178.434,6.460,148.717
C02535=1177.091,147.683,-55.315,-178.431,6.462,148.716
C02536=1177.086,147.932,-55.337,-178.429,6.463,148.716
C02537=1177.082,148.181,-55.357,-178.426,6.464,148.715
C02538=1177.077,148.430,-55.379,-178.423,6.466,148.715
C02539=1177.073,148.679,-55.399,-178.420,6.468,148.714
C02540=1177.068,148.928,-55.421,-178.418,6.470,148.714
C02541=1177.063,149.177,-55.442,-178.415,6.471,148.714
C02542=1177.058,149.426,-55.462,-178.412,6.473,148.713
C02543=1177.053,149.676,-55.483,-178.410,6.475,148.713
C02544=1177.050,149.925,-55.505,-178.407,6.477,148.713
C02545=1177.045,150.174,-55.526,-178.404,6.479,148.712
C02546=1177.039,150.423,-55.547,-178.402,6.480,148.712
C02547=1177.035,150.671,-55.568,-178.399,6.482,148.711
C02548=1177.030,150.921,-55.589,-178.396,6.483,148.711
C02549=1177.025,151.170,-55.610,-178.394,6.484,148.710
C02550=1177.021,151.419,-55.631,-178.391,6.486,148.710
C02551=1177.016,151.668,-55.652,-178.388,6.488,148.710
C02552=1177.011,151.917,-55.674,-178.386,6.490,148.709
C02553=1177.006,152.166,-55.695,-178.383,6.491,148.709
C02554=1177.002,152.415,-55.715,-178.380,6.493,148.709
C02555=1176.997,152.664,-55.737,-178.378,6.495,148.708
C02556=1176.992,152.914,-55.758,-178.375,6.497,148.708
C02557=1176.988,153.162,-55.779,-178.372,6.498,148.707
C02558=1176.983,153.411,-55.800,-178.369,6.500,148.707
C02559=1176.978,153.660,-55.822,-178.367,6.502,148.707
C02560=1176.974,153.910,-55.843,-178.364,6.504,148.706
C02561=1176.969,154.158,-55.864,-178.361,6.505,148.706
C02562=1176.964,154.407,-55.885,-178.359,6.507,148.706
C02563=1176.959,154.656,-55.907,-178.356,6.509,148.705
C02564=1176.955,154.906,-55.928,-178.353,6.510,148.705
C02565=1176.950,155.155,-55.950,-178.351,6.511,148.704
C02566=1176.946,155.404,-55.970,-178.348,6.513,148.704
C02567=1176.941,155.652,-55.992,-178.345,6.515,148.703
C02568=1176.936,155.902,-56.013,-178.343,6.517,148.703
C02569=1176.931,156.151,-56.035,-178.340,6.518,148.703
C02570=1176.926,156.400,-56.056,-178.337,6.520,148.702
C02571=1176.921,156.649,-56.078,-178.335,6.522,148.702
C02572=1176.918,156.898,-56.099,-178.332,6.524,148.702
C02573=1176.912,157.147,-56.120,-178.329,6.525,148.701
C02574=1176.908,157.396,-56.142,-178.327,6.527,148.701
C02575=1176.903,157.646,-56.163,-178.324,6.529,148.700
C02576=1176.898,157.894,-56.185,-178.321,6.531,148.700
C02577=1176.893,158.163,-56.207,-178.318,6.532,148.700
C02578=1176.888,158.432,-56.231,-178.316,6.534,148.699
C02579=1176.883,158.701,-56.254,-178.312,6.536,148.699
C02580=1176.878,158.971,-56.278,-178.309,6.538,148.698
C02581=1176.873,159.219,-56.299,-178.307,6.540,148.698
C02582=1176.868,159.468,-56.321,-178.304,6.542,148.698
C02583=1176.864,159.718,-56.342,-178.301,6.543,148.697
C02584=1176.860,159.966,-56.363,-178.299,6.545,148.697
C02585=1176.855,160.215,-56.385,-178.296,6.547,148.696
C02586=1176.850,160.464,-56.407,-178.293,6.549,148.696
C02587=1176.845,160.713,-56.428,-178.291,6.551,148.696
C02588=1176.840,160.962,-56.450,-178.288,6.552,148.695
C02589=1176.836,161.211,-56.472,-178.285,6.554,148.695
C02590=1176.831,161.460,-56.493,-178.282,6.556,148.695
C02591=1176.827,161.709,-56.516,-178.280,6.558,148.694
C02592=1176.822,161.959,-56.537,-178.277,6.559,148.694
C02593=1176.817,162.207,-56.558,-178.274,6.561,148.693
C02594=1176.813,162.457,-56.580,-178.272,6.563,148.693
C02595=1176.808,162.705,-56.602,-178.269,6.565,148.693
C02596=1176.804,162.955,-56.624,-178.266,6.566,148.692
C02597=1176.799,163.203,-56.646,-178.264,6.568,148.692
C02598=1176.794,163.452,-56.667,-178.261,6.570,148.692
C02599=1176.789,163.701,-56.689,-178.258,6.572,148.691
C02600=1176.785,163.950,-56.711,-178.256,6.573,148.691
C02601=1176.780,164.200,-56.732,-178.253,6.575,148.691
C02602=1176.774,164.449,-56.755,-178.250,6.577,148.690
C02603=1176.770,164.697,-56.776,-178.248,6.579,148.690
C02604=1176.765,164.947,-56.798,-178.245,6.581,148.689
C02605=1176.760,165.195,-56.820,-178.242,6.582,148.689
C02606=1176.756,165.445,-56.842,-178.240,6.584,148.689
C02607=1176.751,165.693,-56.864,-178.237,6.586,148.688
C02608=1176.747,165.943,-56.886,-178.234,6.588,148.688
C02609=1176.742,166.191,-56.908,-178.231,6.589,148.688
C02610=1176.738,166.441,-56.930,-178.229,6.591,148.687
C02611=1176.733,166.689,-56.951,-178.227,6.593,148.687
C02612=1176.728,166.939,-56.974,-178.224,6.595,148.687
C02613=1176.723,167.188,-56.996,-178.221,6.597,148.686
C02614=1176.719,167.436,-57.018,-178.219,6.599,148.686
C02615=1176.714,167.685,-57.040,-178.216,6.600,148.686
C02616=1176.710,167.934,-57.062,-178.213,6.602,148.685
C02617=1176.705,168.183,-57.084,-178.210,6.604,148.685
C02618=1176.700,168.433,-57.106,-178.208,6.606,148.684
C02619=1176.695,168.681,-57.128,-178.205,6.607,148.684
C02620=1176.691,168.931,-57.150,-178.202,6.610,148.684
C02621=1176.686,169.179,-57.172,-178.199,6.612,148.683
C02622=1176.681,169.428,-57.195,-178.196,6.613,148.683
C02623=1176.677,169.677,-57.217,-178.194,6.615,148.683
C02624=1176.672,169.926,-57.239,-178.191,6.617,148.682
C02625=1176.667,170.175,-57.261,-178.188,6.619,148.682
C02626=1176.663,170.424,-57.283,-178.186,6.621,148.682
C02627=1176.658,170.672,-57.306,-178.183,6.622,148.681
C02628=1176.654,170.922,-57.328,-178.180,6.624,148.681
C02629=1176.649,171.170,-57.349,-178.178,6.626,148.680
C02630=1176.644,171.420,-57.372,-178.175,6.628,148.680
C02631=1176.640,171.669,-57.395,-178.173,6.630,148.680
C02632=1176.635,171.917,-57.416,-178.170,6.632,148.680
C02633=1176.631,172.167,-57.439,-178.167,6.633,148.679
C02634=1176.625,172.416,-57.461,-178.165,6.635,148.679
C02635=1176.621,172.664,-57.484,-178.162,6.638,148.679
C02636=1176.617,172.914,-57.506,-178.159,6.639,148.678
C02637=1176.611,173.163,-57.528,-178.156,6.641,148.678
C02638=1176.607,173.412,-57.551,-178.153,6.643,148.677
C02639=1176.602,173.660,-57.572,-178.151,6.645,148.677
C02640=1176.597,173.910,-57.595,-178.148,6.646,148.677
C02641=1176.593,174.159,-57.618,-178.145,6.648,148.676
C02642=1176.588,174.407,-57.640,-178.143,6.650,148.676
C02643=1176.584,174.656,-57.663,-178.141,6.652,148.676
C02644=1176.579,174.905,-57.684,-178.138,6.654,148.675
C02645=1176.574,175.154,-57.707,-178.135,6.656,148.675
C02646=1176.570,175.403,-57.730,-178.133,6.657,148.675
C02647=1176.564,175.652,-57.752,-178.129,6.660,148.674
C02648=1176.560,175.901,-57.775,-178.127,6.662,148.674
C02649=1176.556,176.150,-57.797,-178.124,6.664,148.674
C02650=1176.551,176.399,-57.820,-178.121,6.665,148.673
C02651=1176.547,176.648,-57.842,-178.119,6.667,148.673
C02652=1176.542,176.897,-57.865,-178.116,6.669,148.673
C02653=1176.537,177.146,-57.887,-178.114,6.671,148.672
C02654=1176.532,177.395,-57.910,-178.111,6.673,148.672
C02655=1176.528,177.644,-57.932,-178.108,6.675,148.672
C02656=1176.523,177.892,-57.955,-178.105,6.677,148.671
C02657=1176.518,178.142,-57.977,-178.102,6.679,148.671
C02658=1176.515,178.390,-58.000,-178.100,6.681,148.671
C02659=1176.510,178.640,-58.023,-178.097,6.682,148.670
C02660=1176.504,178.888,-58.046,-178.094,6.684,148.670
C02661=1176.500,179.137,-58.069,-178.092,6.686,148.670
C02662=1176.495,179.387,-58.091,-178.089,6.688,148.669
C02663=1176.491,179.635,-58.114,-178.087,6.690,148.669
C02664=1176.486,179.884,-58.137,-178.084,6.693,148.669
C02665=1176.482,180.133,-58.159,-178.081,6.694,148.668
C02666=1176.477,180.382,-58.182,-178.078,6.696,148.668
C02667=1176.472,180.630,-58.205,-178.076,6.698,148.668
C02668=1176.467,180.880,-58.228,-178.073,6.700,148.667
C02669=1176.463,181.129,-58.250,-178.071,6.702,148.667
C02670=1176.459,181.378,-58.274,-178.068,6.704,148.667
C02671=1176.453,181.626,-58.296,-178.065,6.705,148.666
C02672=1176.449,181.875,-58.319,-178.062,6.708,148.666
C02673=1176.445,182.124,-58.342,-178.059,6.710,148.666
C02674=1176.441,182.373,-58.365,-178.057,6.711,148.665
C02675=1176.435,182.622,-58.387,-178.054,6.713,148.665
C02676=1176.430,182.871,-58.410,-178.052,6.715,148.665
C02677=1176.426,183.120,-58.433,-178.049,6.717,148.665
C02678=1176.422,183.369,-58.457,-178.046,6.719,148.664
C02679=1176.418,183.617,-58.479,-178.043,6.721,148.664
C02680=1176.412,183.866,-58.502,-178.041,6.723,148.663
C02681=1176.407,184.136,-58.527,-178.038,6.725,148.663
C02682=1176.403,184.406,-58.552,-178.035,6.728,148.663
C02683=1176.398,184.675,-58.577,-178.032,6.729,148.662
C02684=1176.392,184.945,-58.602,-178.029,6.731,148.662
C02685=1176.388,185.193,-58.625,-178.026,6.734,148.662
C02686=1176.383,185.442,-58.648,-178.024,6.736,148.662
C02687=1176.378,185.692,-58.671,-178.021,6.738,148.661
C02688=1176.373,185.941,-58.694,-178.018,6.739,148.661
C02689=1176.369,186.190,-58.717,-178.016,6.741,148.661
C02690=1176.365,186.439,-58.740,-178.013,6.744,148.660
C02691=1176.359,186.687,-58.763,-178.010,6.746,148.660
C02692=1176.355,186.936,-58.786,-178.008,6.748,148.660
C02693=1176.351,187.185,-58.809,-178.005,6.750,148.659
C02694=1176.346,187.434,-58.833,-178.002,6.751,148.659
C02695=1176.341,187.683,-58.856,-178.000,6.753,148.659
C02696=1176.337,187.932,-58.879,-177.996,6.756,148.658
C02697=1176.333,188.181,-58.902,-177.994,6.758,148.658
C02698=1176.328,188.430,-58.925,-177.992,6.760,148.658
C02699=1176.323,188.679,-58.949,-177.989,6.761,148.657
C02700=1176.318,188.927,-58.972,-177.986,6.763,148.657
C02701=1176.313,189.176,-58.995,-177.983,6.766,148.657
C02702=1176.309,189.425,-59.018,-177.981,6.768,148.657
C02703=1176.305,189.673,-59.042,-177.978,6.770,148.656
C02704=1176.300,189.922,-59.065,-177.975,6.771,148.656
C02705=1176.296,190.171,-59.089,-177.973,6.773,148.656
C02706=1176.291,190.420,-59.112,-177.969,6.776,148.655
C02707=1176.286,190.669,-59.135,-177.967,6.778,148.655
C02708=1176.281,190.918,-59.159,-177.965,6.780,148.655
C02709=1176.277,191.167,-59.182,-177.962,6.781,148.654
C02710=1176.272,191.416,-59.205,-177.959,6.783,148.654
C02711=1176.268,191.664,-59.229,-177.956,6.786,148.654
C02712=1176.264,191.914,-59.252,-177.954,6.788,148.654
C02713=1176.259,192.163,-59.276,-177.951,6.790,148.653
C02714=1176.254,192.412,-59.299,-177.948,6.792,148.653
C02715=1176.249,192.660,-59.322,-177.946,6.793,148.653
C02716=1176.245,192.908,-59.346,-177.943,6.796,148.652
C02717=1176.240,193.157,-59.369,-177.940,6.798,148.652
C02718=1176.235,193.406,-59.393,-177.938,6.800,148.652
C02719=1176.231,193.655,-59.417,-177.935,6.802,148.651
C02720=1176.226,193.904,-59.440,-177.932,6.805,148.651
C02721=1176.221,194.153,-59.464,-177.930,6.806,148.651
C02722=1176.217,194.402,-59.487,-177.927,6.808,148.651
C02723=1176.212,194.650,-59.511,-177.924,6.810,148.650
C02724=1176.208,194.899,-59.534,-177.922,6.812,148.650
C02725=1176.204,195.149,-59.558,-177.919,6.815,148.650
C02726=1176.199,195.397,-59.582,-177.916,6.816,148.649
C02727=1176.194,195.647,-59.606,-177.913,6.818,148.649
C02728=1176.190,195.896,-59.629,-177.911,6.820,148.649
C02729=1176.185,196.144,-59.653,-177.908,6.823,148.649
C02730=1176.181,196.393,-59.676,-177.905,6.825,148.648
C02731=1176.176,196.641,-59.700,-177.903,6.827,148.648
C02732=1176.172,196.890,-59.724,-177.900,6.828,148.648
C02733=1176.167,197.139,-59.748,-177.897,6.831,148.647
C02734=1176.162,197.388,-59.771,-177.895,6.833,148.647
C02735=1176.158,197.637,-59.795,-177.892,6.835,148.647
C02736=1176.153,197.886,-59.819,-177.890,6.837,148.647
C02737=1176.148,198.135,-59.843,-177.886,6.840,148.646
C02738=1176.144,198.383,-59.867,-177.884,6.841,148.646
C02739=1176.139,198.632,-59.890,-177.881,6.843,148.646
C02740=1176.134,198.881,-59.914,-177.879,6.845,148.646
C02741=1176.130,199.130,-59.938,-177.876,6.848,148.645
C02742=1176.126,199.379,-59.962,-177.873,6.850,148.645
C02743=1176.122,199.627,-59.986,-177.870,6.851,148.644
C02744=1176.116,199.876,-60.010,-177.868,6.854,148.644
C02745=1176.112,200.125,-60.034,-177.865,6.856,148.644
C02746=1176.107,200.374,-60.057,-177.862,6.858,148.644
C02747=1176.103,200.622,-60.081,-177.860,6.860,148.644
C02748=1176.098,200.871,-60.106,-177.857,6.863,148.643
C02749=1176.093,201.121,-60.130,-177.854,6.864,148.643
C02750=1176.089,201.369,-60.154,-177.852,6.866,148.643
C02751=1176.084,201.618,-60.177,-177.849,6.868,148.642
C02752=1176.080,201.867,-60.201,-177.846,6.871,148.642
C02753=1176.076,202.115,-60.225,-177.843,6.873,148.642
C02754=1176.070,202.364,-60.249,-177.841,6.875,148.642
C02755=1176.066,202.613,-60.274,-177.838,6.878,148.641
C02756=1176.062,202.862,-60.298,-177.835,6.879,148.641
C02757=1176.058,203.110,-60.322,-177.833,6.881,148.641
C02758=1176.052,203.360,-60.346,-177.830,6.883,148.641
C02759=1176.048,203.608,-60.370,-177.827,6.886,148.640
C02760=1176.044,203.857,-60.394,-177.825,6.888,148.640
C02761=1176.039,204.106,-60.419,-177.822,6.890,148.640
C02762=1176.034,204.355,-60.442,-177.819,6.892,148.639
C02763=1176.030,204.603,-60.467,-177.816,6.894,148.639
C02764=1176.025,204.852,-60.491,-177.814,6.896,148.639
C02765=1176.021,205.101,-60.516,-177.811,6.899,148.639
C02766=1176.016,205.350,-60.540,-177.808,6.901,148.638
C02767=1176.012,205.599,-60.563,-177.806,6.903,148.638
C02768=1176.007,205.847,-60.588,-177.804,6.905,148.638
C02769=1176.003,206.096,-60.612,-177.800,6.907,148.637
C02770=1175.998,206.345,-60.636,-177.798,6.909,148.637
C02771=1175.993,206.594,-60.661,-177.795,6.911,148.637
C02772=1175.989,206.842,-60.685,-177.792,6.914,148.637
C02773=1175.984,207.091,-60.710,-177.790,6.916,148.637
C02774=1175.980,207.340,-60.734,-177.787,6.918,148.636
C02775=1175.975,207.588,-60.758,-177.784,6.920,148.636
C02776=1175.970,207.837,-60.783,-177.782,6.922,148.636
C02777=1175.966,208.087,-60.807,-177.779,6.924,148.635
C02778=1175.961,208.335,-60.831,-177.776,6.927,148.635
C02779=1175.957,208.584,-60.855,-177.774,6.929,148.635
C02780=1175.952,208.833,-60.880,-177.771,6.931,148.635
C02781=1175.948,209.082,-60.904,-177.768,6.934,148.635
C02782=1175.943,209.330,-60.929,-177.766,6.935,148.634
C02783=1175.938,209.579,-60.953,-177.763,6.937,148.634
C02784=1175.934,209.828,-60.978,-177.760,6.940,148.634
C02785=1175.929,210.098,-61.004,-177.758,6.942,148.633
C02786=1175.924,210.368,-61.031,-177.754,6.945,148.633
C02787=1175.920,210.639,-61.058,-177.751,6.947,148.633
C02788=1175.914,210.909,-61.085,-177.749,6.949,148.633
C02789=1175.909,211.158,-61.110,-177.746,6.952,148.632
C02790=1175.906,211.407,-61.134,-177.743,6.954,148.632
C02791=1175.900,211.656,-61.159,-177.741,6.956,148.632
C02792=1175.896,211.904,-61.183,-177.738,6.958,148.632
C02793=1175.892,212.153,-61.208,-177.735,6.960,148.631
C02794=1175.887,212.402,-61.233,-177.733,6.962,148.631
C02795=1175.882,212.650,-61.257,-177.730,6.965,148.631
C02796=1175.878,212.900,-61.282,-177.727,6.967,148.631
C02797=1175.873,213.148,-61.306,-177.725,6.969,148.630
C02798=1175.869,213.398,-61.331,-177.721,6.972,148.630
C02799=1175.865,213.645,-61.356,-177.719,6.974,148.630
C02800=1175.860,213.894,-61.381,-177.716,6.976,148.630
C02801=1175.856,214.143,-61.405,-177.713,6.978,148.629
C02802=1175.851,214.392,-61.430,-177.711,6.980,148.629
C02803=1175.846,214.641,-61.456,-177.708,6.983,148.629
C02804=1175.842,214.889,-61.480,-177.706,6.985,148.629
C02805=1175.837,215.138,-61.504,-177.703,6.987,148.628
C02806=1175.833,215.387,-61.530,-177.700,6.989,148.628
C02807=1175.828,215.635,-61.554,-177.698,6.992,148.628
C02808=1175.824,215.884,-61.579,-177.694,6.994,148.628
C02809=1175.819,216.133,-61.605,-177.692,6.996,148.628
C02810=1175.815,216.382,-61.629,-177.690,6.998,148.627
C02811=1175.810,216.630,-61.654,-177.687,7.001,148.627
C02812=1175.805,216.878,-61.679,-177.684,7.003,148.627
C02813=1175.801,217.128,-61.704,-177.682,7.005,148.627
C02814=1175.796,217.376,-61.728,-177.679,7.008,148.626
C02815=1175.792,217.625,-61.754,-177.676,7.009,148.626
C02816=1175.787,217.874,-61.779,-177.673,7.012,148.626
C02817=1175.783,218.122,-61.804,-177.671,7.014,148.626
C02818=1175.778,218.371,-61.828,-177.668,7.016,148.625
C02819=1175.774,218.620,-61.854,-177.665,7.019,148.625
C02820=1175.769,218.869,-61.879,-177.663,7.021,148.625
C02821=1175.765,219.117,-61.904,-177.660,7.024,148.625
C02822=1175.760,219.366,-61.929,-177.657,7.025,148.625
C02823=1175.756,219.615,-61.954,-177.655,7.028,148.624
C02824=1175.751,219.863,-61.979,-177.652,7.030,148.624
C02825=1175.747,220.112,-62.004,-177.650,7.032,148.624
C02826=1175.742,220.361,-62.029,-177.646,7.035,148.624
C02827=1175.738,220.609,-62.055,-177.644,7.037,148.623
C02828=1175.734,220.859,-62.080,-177.641,7.040,148.623
C02829=1175.729,221.107,-62.105,-177.638,7.041,148.623
C02830=1175.725,221.356,-62.131,-177.636,7.044,148.623
C02831=1175.720,221.604,-62.155,-177.633,7.046,148.623
C02832=1175.716,221.853,-62.181,-177.631,7.048,148.622
C02833=1175.711,222.102,-62.205,-177.627,7.051,148.622
C02834=1175.707,222.350,-62.231,-177.625,7.053,148.622
C02835=1175.702,222.599,-62.257,-177.622,7.056,148.622
C02836=1175.697,222.848,-62.282,-177.620,7.058,148.622
C02837=1175.693,223.097,-62.307,-177.617,7.060,148.621
C02838=1175.688,223.345,-62.333,-177.614,7.063,148.621
C02839=1175.684,223.594,-62.358,-177.612,7.064,148.621
C02840=1175.680,223.842,-62.383,-177.609,7.067,148.621
C02841=1175.675,224.091,-62.408,-177.606,7.069,148.620
C02842=1175.670,224.339,-62.434,-177.603,7.072,148.620
C02843=1175.666,224.588,-62.459,-177.601,7.074,148.620
C02844=1175.662,224.837,-62.484,-177.598,7.076,148.620
C02845=1175.657,225.085,-62.510,-177.596,7.079,148.620
C02846=1175.653,225.334,-62.536,-177.593,7.081,148.619
C02847=1175.648,225.583,-62.561,-177.590,7.083,148.619
C02848=1175.643,225.832,-62.586,-177.588,7.085,148.619
C02849=1175.639,226.080,-62.612,-177.585,7.088,148.619
C02850=1175.635,226.329,-62.638,-177.582,7.090,148.618
C02851=1175.630,226.577,-62.663,-177.579,7.093,148.618
C02852=1175.626,226.826,-62.689,-177.577,7.095,148.618
C02853=1175.621,227.074,-62.714,-177.574,7.098,148.618
C02854=1175.617,227.323,-62.740,-177.571,7.100,148.618
C02855=1175.612,227.573,-62.765,-177.569,7.102,148.617
C02856=1175.607,227.821,-62.790,-177.566,7.104,148.617
C02857=1175.603,228.069,-62.816,-177.564,7.106,148.617
C02858=1175.598,228.319,-62.842,-177.561,7.109,148.617
C02859=1175.594,228.567,-62.868,-177.558,7.111,148.617
C02860=1175.589,228.815,-62.893,-177.556,7.114,148.617
C02861=1175.585,229.064,-62.919,-177.553,7.116,148.616
C02862=1175.581,229.313,-62.945,-177.550,7.119,148.616
C02863=1175.576,229.561,-62.970,-177.547,7.121,148.616
C02864=1175.572,229.810,-62.996,-177.545,7.124,148.616
C02865=1175.567,230.059,-63.022,-177.542,7.125,148.615
C02866=1175.563,230.307,-63.047,-177.539,7.128,148.615
C02867=1175.558,230.556,-63.073,-177.537,7.130,148.615
C02868=1175.553,230.805,-63.099,-177.534,7.133,148.615
C02869=1175.549,231.054,-63.125,-177.531,7.135,148.615
C02870=1175.544,231.302,-63.150,-177.528,7.138,148.615
C02871=1175.540,231.550,-63.177,-177.526,7.140,148.614
C02872=1175.536,231.799,-63.203,-177.523,7.143,148.614
C02873=1175.531,232.048,-63.229,-177.521,7.145,148.614
C02874=1175.526,232.296,-63.254,-177.518,7.148,148.614
C02875=1175.522,232.545,-63.280,-177.515,7.150,148.614
C02876=1175.518,232.794,-63.306,-177.512,7.152,148.613
C02877=1175.514,233.042,-63.332,-177.510,7.154,148.613
C02878=1175.509,233.291,-63.359,-177.507,7.157,148.613
C02879=1175.504,233.539,-63.384,-177.505,7.159,148.613
C02880=1175.500,233.788,-63.410,-177.502,7.162,148.613
C02881=1175.496,234.037,-63.436,-177.499,7.164,148.612
C02882=1175.491,234.286,-63.462,-177.497,7.167,148.612
C02883=1175.487,234.534,-63.488,-177.494,7.169,148.612
C02884=1175.482,234.782,-63.514,-177.491,7.172,148.612
C02885=1175.478,235.031,-63.540,-177.489,7.174,148.612
C02886=1175.473,235.280,-63.566,-177.486,7.176,148.612
C02887=1175.469,235.528,-63.592,-177.484,7.179,148.611
C02888=1175.465,235.777,-63.618,-177.480,7.181,148.611
C02889=1175.459,236.049,-63.647,-177.478,7.184,148.611
C02890=1175.454,236.320,-63.675,-177.474,7.187,148.611
C02891=1175.450,236.591,-63.704,-177.472,7.189,148.611
C02892=1175.445,236.863,-63.733,-177.469,7.192,148.610
C02893=1175.440,237.112,-63.758,-177.466,7.195,148.610
C02894=1175.436,237.360,-63.785,-177.464,7.197,148.610
C02895=1175.431,237.609,-63.811,-177.461,7.199,148.610
C02896=1175.428,237.857,-63.838,-177.459,7.201,148.610
C02897=1175.422,238.106,-63.864,-177.455,7.204,148.610
C02898=1175.418,238.355,-63.889,-177.453,7.206,148.609
C02899=1175.414,238.603,-63.916,-177.450,7.209,148.609
C02900=1175.409,238.852,-63.942,-177.447,7.212,148.609
C02901=1175.405,239.100,-63.969,-177.445,7.214,148.609
C02902=1175.400,239.349,-63.995,-177.442,7.217,148.609
C02903=1175.396,239.597,-64.021,-177.440,7.219,148.609
C02904=1175.391,239.847,-64.048,-177.437,7.222,148.609
C02905=1175.387,240.095,-64.074,-177.435,7.224,148.608
C02906=1175.383,240.344,-64.100,-177.432,7.226,148.608
C02907=1175.378,240.592,-64.127,-177.429,7.229,148.608
C02908=1175.373,240.840,-64.152,-177.427,7.232,148.608
C02909=1175.369,241.089,-64.179,-177.423,7.234,148.608
C02910=1175.365,241.337,-64.206,-177.421,7.236,148.608
C02911=1175.360,241.586,-64.232,-177.418,7.239,148.608
C02912=1175.356,241.834,-64.259,-177.416,7.241,148.607
C02913=1175.351,242.083,-64.285,-177.413,7.244,148.607
C02914=1175.347,242.331,-64.312,-177.411,7.246,148.607
C02915=1175.343,242.580,-64.339,-177.408,7.249,148.607
C02916=1175.338,242.829,-64.365,-177.405,7.252,148.607
C02917=1175.334,243.077,-64.391,-177.403,7.254,148.607
C02918=1175.329,243.326,-64.418,-177.399,7.257,148.606
C02919=1175.325,243.575,-64.444,-177.397,7.259,148.606
C02920=1175.320,243.823,-64.471,-177.395,7.262,148.606
C02921=1175.316,244.071,-64.498,-177.392,7.263,148.606
C02922=1175.312,244.320,-64.525,-177.389,7.266,148.606
C02923=1175.307,244.569,-64.551,-177.386,7.269,148.606
C02924=1175.303,244.817,-64.578,-177.384,7.271,148.605
C02925=1175.298,245.065,-64.605,-177.381,7.274,148.605
C02926=1175.294,245.314,-64.631,-177.379,7.276,148.605
C02927=1175.289,245.563,-64.657,-177.376,7.279,148.605
C02928=1175.284,245.811,-64.685,-177.373,7.282,148.605
C02929=1175.281,246.059,-64.711,-177.371,7.284,148.605
C02930=1175.276,246.308,-64.738,-177.368,7.287,148.605
C02931=1175.271,246.556,-64.765,-177.365,7.289,148.604
C02932=1175.267,246.805,-64.792,-177.363,7.292,148.604
C02933=1175.263,247.054,-64.818,-177.360,7.295,148.604
C02934=1175.258,247.303,-64.845,-177.358,7.297,148.604
C02935=1175.254,247.551,-64.872,-177.354,7.300,148.604
C02936=1175.250,247.800,-64.899,-177.352,7.302,148.604
C02937=1175.245,248.048,-64.926,-177.349,7.305,148.604
C02938=1175.240,248.297,-64.953,-177.346,7.307,148.603
C02939=1175.236,248.545,-64.979,-177.344,7.309,148.603
C02940=1175.232,248.793,-65.007,-177.341,7.312,148.603
C02941=1175.227,249.042,-65.034,-177.339,7.315,148.603
C02942=1175.222,249.290,-65.061,-177.336,7.317,148.603
C02943=1175.219,249.538,-65.087,-177.333,7.320,148.603
C02944=1175.215,249.788,-65.115,-177.331,7.322,148.603
C02945=1175.210,250.036,-65.142,-177.328,7.325,148.603
C02946=1175.205,250.285,-65.169,-177.325,7.328,148.602
C02947=1175.201,250.533,-65.195,-177.323,7.330,148.602
C02948=1175.197,250.781,-65.222,-177.320,7.333,148.602
C02949=1175.192,251.030,-65.249,-177.317,7.336,148.602
C02950=1175.187,251.278,-65.276,-177.315,7.338,148.602
C02951=1175.183,251.527,-65.303,-177.312,7.341,148.602
C02952=1175.179,251.776,-65.331,-177.309,7.344,148.602
C02953=1175.175,252.024,-65.357,-177.307,7.346,148.602
C02954=1175.170,252.272,-65.385,-177.304,7.349,148.602
C02955=1175.166,252.521,-65.412,-177.302,7.351,148.601
C02956=1175.161,252.769,-65.439,-177.299,7.354,148.601
C02957=1175.157,253.018,-65.467,-177.296,7.357,148.601
C02958=1175.152,253.267,-65.494,-177.294,7.359,148.601
C02959=1175.148,253.515,-65.521,-177.291,7.362,148.601
C02960=1175.143,253.763,-65.549,-177.288,7.364,148.601
C02961=1175.139,254.011,-65.575,-177.286,7.366,148.601
C02962=1175.135,254.261,-65.602,-177.283,7.369,148.601
C02963=1175.131,254.509,-65.629,-177.280,7.372,148.600
C02964=1175.126,254.757,-65.657,-177.278,7.375,148.600
C02965=1175.122,255.005,-65.684,-177.275,7.377,148.600
C02966=1175.117,255.254,-65.711,-177.272,7.380,148.600
C02967=1175.113,255.502,-65.740,-177.270,7.382,148.600
C02968=1175.109,255.751,-65.767,-177.267,7.385,148.600
C02969=1175.104,255.999,-65.794,-177.265,7.388,148.600
C02970=1175.099,256.248,-65.821,-177.262,7.390,148.600
C02971=1175.096,256.497,-65.849,-177.259,7.393,148.599
C02972=1175.091,256.745,-65.876,-177.256,7.396,148.599
C02973=1175.087,256.993,-65.904,-177.254,7.398,148.599
C02974=1175.082,257.241,-65.931,-177.252,7.401,148.599
C02975=1175.078,257.491,-65.958,-177.249,7.404,148.599
C02976=1175.073,257.738,-65.986,-177.246,7.406,148.599
C02977=1175.069,257.987,-66.013,-177.243,7.409,148.599
C02978=1175.065,258.236,-66.041,-177.241,7.412,148.599
C02979=1175.060,258.484,-66.068,-177.238,7.414,148.599
C02980=1175.056,258.732,-66.096,-177.236,7.417,148.599
C02981=1175.051,258.980,-66.123,-177.233,7.420,148.599
C02982=1175.047,259.229,-66.152,-177.231,7.422,148.599
C02983=1175.042,259.478,-66.179,-177.228,7.425,148.598
C02984=1175.038,259.726,-66.207,-177.225,7.428,148.598
C02985=1175.034,259.975,-66.234,-177.222,7.431,148.598
C02986=1175.029,260.223,-66.262,-177.220,7.433,148.598
C02987=1175.025,260.471,-66.289,-177.217,7.436,148.598
C02988=1175.021,260.720,-66.317,-177.214,7.439,148.598
C02989=1175.016,260.968,-66.344,-177.212,7.441,148.598
C02990=1175.011,261.216,-66.372,-177.210,7.444,148.598
C02991=1175.007,261.466,-66.400,-177.206,7.447,148.598
C02992=1175.003,261.714,-66.428,-177.204,7.449,148.597
C02993=1174.998,261.987,-66.458,-177.201,7.452,148.597
C02994=1174.993,262.260,-66.489,-177.198,7.455,148.597
C02995=1174.988,262.533,-66.519,-177.195,7.458,148.597
C02996=1174.984,262.806,-66.550,-177.192,7.461,148.597
C02997=1174.979,263.054,-66.578,-177.189,7.464,148.597
C02998=1174.976,263.303,-66.606,-177.187,7.466,148.597
C02999=1174.971,263.551,-66.633,-177.185,7.469,148.597
C03000=1174.967,263.799,-66.661,-177.182,7.472,148.597
C03001=1174.962,264.048,-66.690,-177.180,7.474,148.597
C03002=1174.958,264.296,-66.717,-177.177,7.477,148.597
C03003=1174.954,264.545,-66.745,-177.174,7.480,148.597
C03004=1174.949,264.793,-66.773,-177.171,7.483,148.597
C03005=1174.944,265.041,-66.801,-177.169,7.485,148.596
C03006=1174.940,265.290,-66.829,-177.166,7.488,148.596
C03007=1174.936,265.538,-66.856,-177.163,7.491,148.596
C03008=1174.931,265.787,-66.885,-177.161,7.493,148.596
C03009=1174.927,266.035,-66.913,-177.158,7.496,148.596
C03010=1174.923,266.283,-66.941,-177.156,7.499,148.596
C03011=1174.918,266.532,-66.969,-177.153,7.502,148.596
C03012=1174.914,266.779,-66.997,-177.151,7.504,148.596
C03013=1174.910,267.028,-67.025,-177.148,7.507,148.596
C03014=1174.905,267.276,-67.053,-177.145,7.510,148.596
C03015=1174.901,267.525,-67.081,-177.142,7.513,148.596
C03016=1174.896,267.774,-67.109,-177.140,7.515,148.596
C03017=1174.892,268.022,-67.137,-177.138,7.518,148.596
C03018=1174.888,268.270,-67.165,-177.135,7.521,148.595
C03019=1174.883,268.519,-67.194,-177.132,7.524,148.595
C03020=1174.879,268.767,-67.222,-177.130,7.526,148.595
C03021=1174.874,269.016,-67.250,-177.127,7.529,148.595
C03022=1174.870,269.264,-67.278,-177.124,7.532,148.595
C03023=1174.866,269.512,-67.306,-177.122,7.535,148.595
C03024=1174.861,269.760,-67.335,-177.119,7.537,148.595
C03025=1174.857,270.009,-67.363,-177.116,7.540,148.595
C03026=1174.852,270.257,-67.391,-177.114,7.543,148.595
C03027=1174.849,270.506,-67.419,-177.111,7.546,148.595
C03028=1174.844,270.755,-67.448,-177.109,7.548,148.595
C03029=1174.840,271.002,-67.477,-177.106,7.551,148.595
C03030=1174.836,271.251,-67.505,-177.103,7.554,148.595
C03031=1174.831,271.499,-67.533,-177.100,7.557,148.595
C03032=1174.827,271.748,-67.562,-177.098,7.560,148.594
C03033=1174.822,271.995,-67.590,-177.095,7.562,148.594
C03034=1174.818,272.244,-67.618,-177.093,7.565,148.594
C03035=1174.814,272.493,-67.646,-177.090,7.568,148.594
C03036=1174.809,272.740,-67.676,-177.087,7.571,148.594
C03037=1174.806,272.989,-67.704,-177.085,7.573,148.594
C03038=1174.801,273.237,-67.732,-177.082,7.576,148.594
C03039=1174.797,273.486,-67.760,-177.080,7.579,148.594
C03040=1174.792,273.735,-67.789,-177.077,7.582,148.594
C03041=1174.788,273.982,-67.818,-177.074,7.585,148.594
C03042=1174.784,274.231,-67.846,-177.072,7.587,148.594
C03043=1174.779,274.479,-67.875,-177.069,7.590,148.594
C03044=1174.775,274.727,-67.903,-177.066,7.593,148.594
C03045=1174.771,274.976,-67.932,-177.064,7.596,148.594
C03046=1174.766,275.224,-67.961,-177.061,7.599,148.594
C03047=1174.762,275.473,-67.989,-177.059,7.601,148.594
C03048=1174.758,275.721,-68.018,-177.056,7.604,148.594
C03049=1174.753,275.969,-68.046,-177.053,7.607,148.594
C03050=1174.749,276.217,-68.075,-177.051,7.611,148.594
C03051=1174.745,276.466,-68.104,-177.048,7.614,148.594
C03052=1174.740,276.714,-68.132,-177.046,7.616,148.594
C03053=1174.736,276.962,-68.161,-177.043,7.619,148.594
C03054=1174.732,277.211,-68.190,-177.041,7.622,148.594
C03055=1174.727,277.458,-68.219,-177.038,7.625,148.593
C03056=1174.723,277.707,-68.247,-177.035,7.628,148.593
C03057=1174.719,277.955,-68.277,-177.033,7.630,148.593
C03058=1174.714,278.204,-68.305,-177.030,7.633,148.593
C03059=1174.710,278.452,-68.333,-177.028,7.636,148.593
C03060=1174.706,278.700,-68.363,-177.025,7.639,148.593
C03061=1174.701,278.949,-68.391,-177.022,7.642,148.593
C03062=1174.697,279.197,-68.421,-177.020,7.644,148.593
C03063=1174.693,279.445,-68.449,-177.017,7.647,148.593
C03064=1174.689,279.694,-68.478,-177.014,7.650,148.593
C03065=1174.684,279.941,-68.507,-177.012,7.653,148.593
C03066=1174.679,280.190,-68.536,-177.009,7.656,148.593
C03067=1174.675,280.438,-68.565,-177.006,7.659,148.593
C03068=1174.672,280.687,-68.594,-177.005,7.661,148.593
C03069=1174.667,280.935,-68.623,-177.002,7.664,148.593
C03070=1174.663,281.183,-68.652,-176.999,7.667,148.593
C03071=1174.658,281.432,-68.681,-176.996,7.670,148.593
C03072=1174.654,281.680,-68.710,-176.994,7.673,148.593
C03073=1174.650,281.928,-68.740,-176.991,7.675,148.593
C03074=1174.645,282.176,-68.768,-176.989,7.678,148.593
C03075=1174.641,282.424,-68.797,-176.986,7.681,148.593
C03076=1174.637,282.673,-68.826,-176.983,7.684,148.593
C03077=1174.633,282.922,-68.855,-176.980,7.687,148.593
C03078=1174.628,283.169,-68.884,-176.978,7.690,148.593
C03079=1174.624,283.417,-68.914,-176.975,7.693,148.593
C03080=1174.619,283.666,-68.943,-176.973,7.696,148.593
C03081=1174.615,283.914,-68.972,-176.971,7.699,148.593
C03082=1174.611,284.163,-69.001,-176.968,7.702,148.593
C03083=1174.607,284.411,-69.031,-176.965,7.704,148.593
C03084=1174.602,284.659,-69.060,-176.962,7.707,148.593
C03085=1174.598,284.907,-69.089,-176.960,7.710,148.593
C03086=1174.594,285.155,-69.117,-176.957,7.713,148.592
C03087=1174.590,285.404,-69.147,-176.955,7.716,148.592
C03088=1174.585,285.652,-69.176,-176.952,7.719,148.593
C03089=1174.581,285.900,-69.206,-176.950,7.722,148.593
C03090=1174.577,286.148,-69.235,-176.947,7.725,148.593
C03091=1174.572,286.396,-69.264,-176.944,7.728,148.593
C03092=1174.568,286.644,-69.294,-176.941,7.731,148.592
C03093=1174.564,286.893,-69.323,-176.939,7.733,148.592
C03094=1174.560,287.141,-69.353,-176.937,7.736,148.592
C03095=1174.555,287.389,-69.383,-176.934,7.739,148.593
C03096=1174.550,287.638,-69.412,-176.932,7.742,148.593
C03097=1174.546,287.912,-69.444,-176.929,7.745,148.592
C03098=1174.541,288.187,-69.476,-176.925,7.749,148.592
C03099=1174.536,288.462,-69.510,-176.923,7.752,148.592
C03100=1174.531,288.737,-69.541,-176.920,7.755,148.592
C03101=1174.527,288.985,-69.571,-176.917,7.758,148.592
C03102=1174.523,289.233,-69.600,-176.915,7.761,148.592
C03103=1174.518,289.482,-69.630,-176.912,7.764,148.592
C03104=1174.514,289.729,-69.661,-176.910,7.767,148.592
C03105=1174.510,289.978,-69.690,-176.907,7.770,148.592
C03106=1174.506,290.226,-69.719,-176.905,7.772,148.592
C03107=1174.502,290.474,-69.749,-176.902,7.775,148.592
C03108=1174.498,290.722,-69.778,-176.899,7.778,148.592
C03109=1174.493,290.971,-69.808,-176.896,7.781,148.592
C03110=1174.488,291.219,-69.838,-176.894,7.785,148.592
C03111=1174.484,291.468,-69.867,-176.891,7.788,148.592
C03112=1174.480,291.715,-69.898,-176.889,7.791,148.592
C03113=1174.476,291.963,-69.927,-176.886,7.794,148.592
C03114=1174.472,292.212,-69.956,-176.884,7.796,148.592
C03115=1174.468,292.460,-69.986,-176.882,7.799,148.592
C03116=1174.463,292.709,-70.016,-176.879,7.802,148.592
C03117=1174.459,292.956,-70.046,-176.876,7.805,148.592
C03118=1174.455,293.204,-70.076,-176.873,7.808,148.592
C03119=1174.451,293.453,-70.105,-176.871,7.811,148.592
C03120=1174.446,293.701,-70.136,-176.868,7.814,148.593
C03121=1174.442,293.949,-70.165,-176.866,7.817,148.593
C03122=1174.438,294.197,-70.195,-176.863,7.820,148.592
C03123=1174.434,294.446,-70.224,-176.860,7.823,148.592
C03124=1174.429,294.693,-70.255,-176.858,7.825,148.592
C03125=1174.425,294.942,-70.284,-176.856,7.829,148.593
C03126=1174.421,295.189,-70.314,-176.853,7.832,148.593
C03127=1174.416,295.438,-70.345,-176.850,7.835,148.593
C03128=1174.412,295.686,-70.374,-176.847,7.838,148.592
C03129=1174.408,295.934,-70.404,-176.845,7.841,148.593
C03130=1174.403,296.182,-70.434,-176.842,7.844,148.593
C03131=1174.400,296.431,-70.465,-176.840,7.847,148.593
C03132=1174.396,296.679,-70.494,-176.837,7.850,148.593
C03133=1174.391,296.928,-70.524,-176.835,7.853,148.593
C03134=1174.387,297.175,-70.554,-176.832,7.856,148.593
C03135=1174.383,297.424,-70.584,-176.830,7.858,148.593
C03136=1174.378,297.672,-70.615,-176.827,7.861,148.593
C03137=1174.374,297.920,-70.644,-176.825,7.864,148.593
C03138=1174.370,298.167,-70.674,-176.822,7.867,148.593
C03139=1174.365,298.415,-70.705,-176.819,7.870,148.593
C03140=1174.361,298.664,-70.734,-176.817,7.873,148.593
C03141=1174.357,298.912,-70.766,-176.814,7.877,148.593
C03142=1174.353,299.161,-70.795,-176.812,7.880,148.593
C03143=1174.348,299.409,-70.826,-176.809,7.883,148.593
C03144=1174.344,299.657,-70.855,-176.806,7.886,148.593
C03145=1174.340,299.905,-70.886,-176.804,7.889,148.593
C03146=1174.336,300.152,-70.916,-176.801,7.892,148.593
C03147=1174.331,300.401,-70.946,-176.798,7.895,148.593
C03148=1174.327,300.649,-70.977,-176.796,7.897,148.593
C03149=1174.323,300.897,-71.008,-176.794,7.900,148.593
C03150=1174.319,301.146,-71.037,-176.791,7.903,148.593
C03151=1174.314,301.394,-71.068,-176.788,7.906,148.593
C03152=1174.310,301.641,-71.098,-176.786,7.910,148.593
C03153=1174.306,301.890,-71.128,-176.783,7.913,148.593
C03154=1174.302,302.138,-71.159,-176.781,7.916,148.593
C03155=1174.297,302.386,-71.189,-176.778,7.919,148.593
C03156=1174.293,302.634,-71.219,-176.776,7.922,148.593
C03157=1174.289,302.882,-71.250,-176.773,7.925,148.593
C03158=1174.285,303.130,-71.280,-176.770,7.928,148.593
C03159=1174.281,303.379,-71.311,-176.768,7.931,148.594
C03160=1174.276,303.627,-71.342,-176.765,7.934,148.593
C03161=1174.272,303.874,-71.372,-176.763,7.937,148.593
C03162=1174.268,304.122,-71.403,-176.760,7.940,148.594
C03163=1174.264,304.371,-71.432,-176.757,7.943,148.594
C03164=1174.259,304.619,-71.463,-176.755,7.946,148.594
C03165=1174.255,304.867,-71.494,-176.752,7.950,148.594
C03166=1174.251,305.115,-71.524,-176.750,7.952,148.594
C03167=1174.247,305.363,-71.555,-176.748,7.955,148.594
C03168=1174.242,305.611,-71.586,-176.745,7.958,148.594
C03169=1174.238,305.859,-71.616,-176.743,7.961,148.594
C03170=1174.234,306.107,-71.647,-176.740,7.964,148.594
C03171=1174.230,306.356,-71.678,-176.738,7.967,148.594
C03172=1174.226,306.603,-71.708,-176.735,7.970,148.594
C03173=1174.221,306.851,-71.739,-176.732,7.973,148.594
C03174=1174.217,307.099,-71.770,-176.730,7.977,148.594
C03175=1174.213,307.348,-71.801,-176.727,7.980,148.594
C03176=1174.209,307.595,-71.831,-176.724,7.983,148.594
C03177=1174.204,307.843,-71.862,-176.722,7.986,148.594
C03178=1174.200,308.092,-71.893,-176.719,7.989,148.594
C03179=1174.196,308.340,-71.924,-176.717,7.992,148.595
C03180=1174.192,308.588,-71.954,-176.714,7.995,148.595
C03181=1174.188,308.836,-71.985,-176.712,7.998,148.594
C03182=1174.183,309.084,-72.016,-176.709,8.002,148.595
C03183=1174.178,309.332,-72.046,-176.707,8.005,148.595
C03184=1174.174,309.581,-72.078,-176.704,8.008,148.595
C03185=1174.171,309.829,-72.108,-176.702,8.011,148.595
C03186=1174.166,310.076,-72.139,-176.699,8.014,148.595
C03187=1174.162,310.325,-72.170,-176.697,8.017,148.595
C03188=1174.158,310.572,-72.201,-176.694,8.020,148.595
C03189=1174.153,310.820,-72.232,-176.691,8.023,148.595
C03190=1174.150,311.069,-72.262,-176.689,8.026,148.595
C03191=1174.145,311.316,-72.294,-176.686,8.029,148.595
C03192=1174.141,311.565,-72.325,-176.684,8.033,148.595
C03193=1174.137,311.813,-72.356,-176.681,8.036,148.595
C03194=1174.132,312.061,-72.387,-176.678,8.039,148.595
C03195=1174.128,312.309,-72.418,-176.676,8.042,148.596
C03196=1174.124,312.557,-72.449,-176.673,8.045,148.595
C03197=1174.120,312.805,-72.480,-176.671,8.048,148.596
C03198=1174.116,313.053,-72.512,-176.668,8.051,148.596
C03199=1174.112,313.300,-72.542,-176.666,8.054,148.596
C03200=1174.108,313.549,-72.573,-176.663,8.057,148.596
C03201=1174.103,313.826,-72.608,-176.661,8.060,148.596
C03202=1174.098,314.103,-72.644,-176.658,8.065,148.596
C03203=1174.093,314.380,-72.677,-176.655,8.068,148.596
C03204=1174.088,314.657,-72.713,-176.652,8.071,148.596
C03205=1174.084,314.904,-72.744,-176.650,8.075,148.596
C03206=1174.080,315.153,-72.775,-176.647,8.078,148.596
C03207=1174.076,315.400,-72.807,-176.645,8.081,148.596
C03208=1174.072,315.649,-72.838,-176.642,8.084,148.596
C03209=1174.067,315.897,-72.869,-176.640,8.087,148.597
C03210=1174.063,316.145,-72.901,-176.637,8.090,148.597
C03211=1174.059,316.393,-72.931,-176.635,8.094,148.597
C03212=1174.055,316.641,-72.963,-176.632,8.097,148.597
C03213=1174.051,316.888,-72.995,-176.629,8.100,148.597
C03214=1174.047,317.137,-73.026,-176.627,8.103,148.597
C03215=1174.042,317.384,-73.057,-176.624,8.106,148.597
C03216=1174.038,317.633,-73.088,-176.622,8.109,148.597
C03217=1174.034,317.880,-73.120,-176.619,8.112,148.597
C03218=1174.030,318.129,-73.151,-176.617,8.115,148.597
C03219=1174.026,318.376,-73.182,-176.614,8.118,148.597
C03220=1174.022,318.624,-73.214,-176.612,8.122,148.598
C03221=1174.018,318.872,-73.245,-176.609,8.125,148.598
C03222=1174.013,319.120,-73.278,-176.607,8.128,148.598
C03223=1174.009,319.368,-73.309,-176.604,8.131,148.598
C03224=1174.005,319.616,-73.340,-176.602,8.134,148.598
C03225=1174.001,319.864,-73.372,-176.599,8.137,148.598
C03226=1173.997,320.112,-73.403,-176.597,8.141,148.598
C03227=1173.993,320.360,-73.435,-176.594,8.144,148.598
C03228=1173.988,320.608,-73.466,-176.592,8.147,148.598
C03229=1173.984,320.856,-73.499,-176.589,8.150,148.598
C03230=1173.980,321.104,-73.530,-176.587,8.153,148.599
C03231=1173.976,321.352,-73.561,-176.584,8.156,148.599
C03232=1173.972,321.600,-73.593,-176.582,8.159,148.599
C03233=1173.968,321.847,-73.624,-176.579,8.163,148.599
C03234=1173.963,322.096,-73.657,-176.577,8.166,148.599
C03235=1173.960,322.344,-73.689,-176.574,8.169,148.599
C03236=1173.955,322.592,-73.719,-176.572,8.172,148.599
C03237=1173.951,322.840,-73.751,-176.569,8.175,148.599
C03238=1173.947,323.088,-73.783,-176.567,8.178,148.599
C03239=1173.942,323.335,-73.815,-176.564,8.182,148.599
C03240=1173.939,323.583,-73.847,-176.562,8.185,148.599
C03241=1173.934,323.831,-73.879,-176.559,8.188,148.600
C03242=1173.931,324.079,-73.910,-176.557,8.191,148.600
C03243=1173.926,324.327,-73.943,-176.554,8.195,148.600
C03244=1173.922,324.575,-73.974,-176.552,8.198,148.600
C03245=1173.918,324.823,-74.006,-176.549,8.201,148.600
C03246=1173.914,325.071,-74.039,-176.547,8.205,148.600
C03247=1173.910,325.318,-74.070,-176.544,8.208,148.600
C03248=1173.906,325.566,-74.102,-176.542,8.211,148.600
C03249=1173.901,325.815,-74.134,-176.539,8.214,148.601
C03250=1173.898,326.063,-74.166,-176.537,8.217,148.601
C03251=1173.893,326.310,-74.198,-176.534,8.221,148.601
C03252=1173.889,326.558,-74.230,-176.532,8.224,148.601
C03253=1173.885,326.806,-74.262,-176.529,8.227,148.601
C03254=1173.880,327.054,-74.294,-176.527,8.230,148.601
C03255=1173.876,327.302,-74.326,-176.524,8.233,148.601
C03256=1173.873,327.550,-74.358,-176.522,8.236,148.601
C03257=1173.868,327.798,-74.390,-176.520,8.240,148.602
C03258=1173.864,328.046,-74.422,-176.517,8.243,148.602
C03259=1173.860,328.294,-74.454,-176.515,8.246,148.602
C03260=1173.856,328.542,-74.487,-176.512,8.250,148.602
C03261=1173.851,328.789,-74.519,-176.509,8.253,148.602
C03262=1173.847,329.037,-74.551,-176.507,8.256,148.602
C03263=1173.844,329.285,-74.582,-176.505,8.260,148.603
C03264=1173.839,329.534,-74.615,-176.502,8.263,148.603
C03265=1173.835,329.780,-74.647,-176.500,8.266,148.603
C03266=1173.831,330.029,-74.680,-176.497,8.269,148.603
C03267=1173.827,330.277,-74.711,-176.495,8.272,148.603
C03268=1173.823,330.525,-74.744,-176.492,8.276,148.603
C03269=1173.819,330.773,-74.777,-176.490,8.279,148.603
C03270=1173.814,331.020,-74.808,-176.487,8.282,148.603
C03271=1173.810,331.269,-74.841,-176.485,8.285,148.604
C03272=1173.806,331.516,-74.873,-176.483,8.289,148.604
C03273=1173.802,331.764,-74.906,-176.479,8.292,148.604
C03274=1173.798,332.012,-74.938,-176.477,8.296,148.604
C03275=1173.793,332.259,-74.971,-176.475,8.299,148.604
C03276=1173.790,332.507,-75.002,-176.472,8.302,148.604
C03277=1173.785,332.756,-75.035,-176.470,8.305,148.604
C03278=1173.781,333.003,-75.068,-176.468,8.309,148.605
C03279=1173.777,333.252,-75.100,-176.465,8.312,148.605
C03280=1173.773,333.499,-75.133,-176.463,8.315,148.605
C03281=1173.769,333.747,-75.164,-176.460,8.318,148.605
C03282=1173.765,333.994,-75.198,-176.458,8.321,148.605
C03283=1173.760,334.243,-75.230,-176.456,8.325,148.605
C03284=1173.757,334.491,-75.262,-176.453,8.329,148.606
C03285=1173.753,334.738,-75.295,-176.450,8.332,148.606
C03286=1173.748,334.987,-75.327,-176.448,8.335,148.606
C03287=1173.745,335.234,-75.360,-176.446,8.338,148.606
C03288=1173.740,335.481,-75.393,-176.443,8.341,148.606
C03289=1173.736,335.730,-75.425,-176.441,8.345,148.606
C03290=1173.732,335.977,-75.458,-176.438,8.348,148.607
C03291=1173.728,336.225,-75.490,-176.436,8.351,148.607
C03292=1173.724,336.473,-75.523,-176.433,8.354,148.607
C03293=1173.720,336.721,-75.555,-176.431,8.358,148.607
C03294=1173.716,336.969,-75.588,-176.428,8.362,148.607
C03295=1173.712,337.217,-75.622,-176.426,8.365,148.607
C03296=1173.707,337.465,-75.654,-176.424,8.368,148.608
C03297=1173.704,337.712,-75.687,-176.421,8.371,148.608
C03298=1173.700,337.960,-75.720,-176.419,8.375,148.608
C03299=1173.695,338.208,-75.752,-176.416,8.378,148.608
C03300=1173.690,338.455,-75.785,-176.414,8.381,148.608
C03301=1173.686,338.703,-75.818,-176.412,8.385,148.608
C03302=1173.683,338.951,-75.850,-176.409,8.389,148.609
C03303=1173.678,339.199,-75.883,-176.406,8.392,148.609
C03304=1173.674,339.447,-75.916,-176.404,8.395,148.609
C03305=1173.670,339.726,-75.954,-176.402,8.398,148.609
C03306=1173.665,340.005,-75.990,-176.399,8.402,148.609
C03307=1173.661,340.284,-76.028,-176.396,8.407,148.610
C03308=1173.656,340.565,-76.065,-176.394,8.410,148.610
C03309=1173.652,340.812,-76.097,-176.391,8.414,148.610
C03310=1173.648,341.060,-76.130,-176.388,8.417,148.610
C03311=1173.644,341.307,-76.164,-176.386,8.420,148.610
C03312=1173.640,341.555,-76.197,-176.384,8.424,148.611
C03313=1173.636,341.803,-76.230,-176.381,8.427,148.611
C03314=1173.632,342.051,-76.263,-176.379,8.430,148.611
C03315=1173.628,342.298,-76.296,-176.377,8.434,148.611
C03316=1173.623,342.547,-76.329,-176.374,8.438,148.611
C03317=1173.619,342.794,-76.362,-176.372,8.441,148.612
C03318=1173.615,343.042,-76.395,-176.369,8.444,148.612
C03319=1173.611,343.290,-76.428,-176.367,8.448,148.612
C03320=1173.607,343.538,-76.461,-176.365,8.451,148.612
C03321=1173.602,343.785,-76.494,-176.363,8.454,148.613
C03322=1173.598,344.033,-76.528,-176.360,8.457,148.613
C03323=1173.594,344.281,-76.561,-176.357,8.461,148.613
C03324=1173.590,344.529,-76.594,-176.355,8.465,148.613
C03325=1173.586,344.776,-76.627,-176.352,8.468,148.613
C03326=1173.582,345.024,-76.660,-176.350,8.471,148.613
C03327=1173.578,345.272,-76.693,-176.348,8.474,148.614
C03328=1173.574,345.519,-76.727,-176.346,8.478,148.614
C03329=1173.570,345.767,-76.760,-176.343,8.482,148.614
C03330=1173.565,346.014,-76.794,-176.341,8.485,148.614
C03331=1173.562,346.263,-76.827,-176.338,8.489,148.615
C03332=1173.558,346.510,-76.860,-176.336,8.492,148.615
C03333=1173.554,346.758,-76.893,-176.334,8.495,148.615
C03334=1173.550,347.006,-76.927,-176.331,8.498,148.615
C03335=1173.545,347.254,-76.960,-176.329,8.503,148.616
C03336=1173.542,347.501,-76.994,-176.327,8.506,148.616
C03337=1173.537,347.748,-77.027,-176.324,8.509,148.616
C03338=1173.533,347.996,-77.060,-176.322,8.513,148.616
C03339=1173.529,348.245,-77.094,-176.320,8.516,148.617
C03340=1173.525,348.492,-77.128,-176.318,8.519,148.617
C03341=1173.521,348.740,-77.161,-176.315,8.524,148.617
C03342=1173.517,348.988,-77.194,-176.313,8.527,148.617
C03343=1173.513,349.235,-77.227,-176.310,8.530,148.617
C03344=1173.509,349.482,-77.261,-176.308,8.533,148.618
C03345=1173.504,349.730,-77.295,-176.306,8.537,148.618
C03346=1173.501,349.979,-77.329,-176.303,8.540,148.618
C03347=1173.497,350.226,-77.362,-176.301,8.544,148.618
C03348=1173.493,350.474,-77.396,-176.299,8.548,148.619
C03349=1173.488,350.721,-77.429,-176.296,8.551,148.619
C03350=1173.485,350.969,-77.463,-176.294,8.554,148.619
C03351=1173.480,351.217,-77.497,-176.292,8.558,148.619
C03352=1173.476,351.464,-77.531,-176.289,8.562,148.620
C03353=1173.472,351.712,-77.564,-176.287,8.565,148.620
C03354=1173.468,351.960,-77.597,-176.284,8.568,148.620
C03355=1173.464,352.207,-77.631,-176.283,8.572,148.621
C03356=1173.460,352.456,-77.665,-176.280,8.575,148.621
C03357=1173.456,352.703,-77.699,-176.278,8.579,148.621
C03358=1173.452,352.951,-77.732,-176.275,8.583,148.621
C03359=1173.448,353.198,-77.766,-176.273,8.586,148.622
C03360=1173.444,353.446,-77.800,-176.271,8.590,148.622
C03361=1173.440,353.693,-77.834,-176.269,8.593,148.622
C03362=1173.435,353.942,-77.867,-176.266,8.597,148.622
C03363=1173.431,354.189,-77.901,-176.264,8.600,148.623
C03364=1173.428,354.436,-77.936,-176.262,8.604,148.623
C03365=1173.423,354.684,-77.969,-176.260,8.607,148.623
C03366=1173.420,354.932,-78.003,-176.257,8.611,148.624
C03367=1173.416,355.180,-78.037,-176.254,8.615,148.624
C03368=1173.411,355.427,-78.071,-176.253,8.618,148.624
C03369=1173.408,355.675,-78.105,-176.250,8.622,148.624
C03370=1173.403,355.922,-78.138,-176.248,8.625,148.625
C03371=1173.399,356.170,-78.173,-176.246,8.629,148.625
C03372=1173.396,356.418,-78.207,-176.243,8.633,148.625
C03373=1173.391,356.666,-78.241,-176.241,8.636,148.626
C03374=1173.388,356.913,-78.275,-176.239,8.639,148.626
C03375=1173.384,357.160,-78.309,-176.236,8.644,148.626
C03376=1173.379,357.409,-78.343,-176.234,8.647,148.626
C03377=1173.376,357.656,-78.377,-176.232,8.650,148.627
C03378=1173.371,357.904,-78.411,-176.230,8.654,148.627
C03379=1173.367,358.151,-78.445,-176.227,8.658,148.627
C03380=1173.363,358.399,-78.480,-176.225,8.662,148.628
C03381=1173.359,358.647,-78.513,-176.223,8.665,148.628
C03382=1173.355,358.895,-78.548,-176.221,8.668,148.628
C03383=1173.351,359.142,-78.582,-176.219,8.672,148.629
C03384=1173.347,359.389,-78.616,-176.216,8.676,148.629
C03385=1173.343,359.637,-78.651,-176.214,8.680,148.629
C03386=1173.339,359.885,-78.685,-176.212,8.683,148.630
C03387=1173.335,360.132,-78.718,-176.210,8.687,148.630
C03388=1173.331,360.380,-78.753,-176.207,8.691,148.630
C03389=1173.327,360.628,-78.787,-176.205,8.694,148.631
C03390=1173.323,360.876,-78.822,-176.203,8.698,148.631
C03391=1173.319,361.123,-78.856,-176.201,8.701,148.631
C03392=1173.315,361.371,-78.890,-176.199,8.705,148.632
C03393=1173.311,361.618,-78.924,-176.197,8.709,148.632
C03394=1173.307,361.865,-78.959,-176.194,8.712,148.632
C03395=1173.304,362.113,-78.993,-176.193,8.716,148.633
C03396=1173.299,362.361,-79.027,-176.191,8.720,148.633
C03397=1173.295,362.609,-79.062,-176.188,8.724,148.633
C03398=1173.291,362.856,-79.096,-176.186,8.727,148.634
C03399=1173.287,363.104,-79.131,-176.184,8.731,148.634
C03400=1173.283,363.351,-79.165,-176.182,8.734,148.635
C03401=1173.279,363.599,-79.200,-176.180,8.738,148.635
C03402=1173.275,363.847,-79.234,-176.178,8.741,148.635
C03403=1173.271,364.094,-79.268,-176.175,8.746,148.636
C03404=1173.267,364.341,-79.304,-176.174,8.749,148.636
C03405=1173.263,364.589,-79.338,-176.172,8.753,148.636
C03406=1173.260,364.836,-79.372,-176.170,8.756,148.637
C03407=1173.255,365.084,-79.407,-176.168,8.760,148.637
C03408=1173.251,365.332,-79.442,-176.166,8.763,148.638
C03409=1173.247,365.613,-79.480,-176.163,8.768,148.638
C03410=1173.243,365.896,-79.520,-176.161,8.772,148.639
C03411=1173.238,366.177,-79.560,-176.159,8.777,148.639
C03412=1173.233,366.460,-79.599,-176.157,8.780,148.639
C03413=1173.229,366.707,-79.634,-176.155,8.784,148.640
C03414=1173.226,366.955,-79.668,-176.153,8.787,148.640
C03415=1173.221,367.202,-79.703,-176.151,8.791,148.641
C03416=1173.217,367.450,-79.738,-176.149,8.795,148.641
C03417=1173.213,367.697,-79.773,-176.147,8.799,148.642
C03418=1173.210,367.945,-79.807,-176.145,8.803,148.642
C03419=1173.205,368.192,-79.842,-176.144,8.807,148.643
C03420=1173.201,368.440,-79.877,-176.142,8.810,148.643
C03421=1173.197,368.687,-79.911,-176.140,8.814,148.644
C03422=1173.193,368.935,-79.947,-176.138,8.817,148.644
C03423=1173.190,369.183,-79.981,-176.136,8.821,148.644
C03424=1173.185,369.430,-80.016,-176.134,8.825,148.645
C03425=1173.182,369.678,-80.051,-176.133,8.829,148.645
C03426=1173.177,369.925,-80.086,-176.131,8.832,148.646
C03427=1173.173,370.173,-80.120,-176.129,8.836,148.646
C03428=1173.169,370.420,-80.156,-176.128,8.839,148.647
C03429=1173.166,370.668,-80.190,-176.126,8.843,148.647
C03430=1173.162,370.915,-80.225,-176.124,8.847,148.648
C03431=1173.157,371.163,-80.260,-176.122,8.850,148.648
C03432=1173.154,371.410,-80.295,-176.121,8.854,148.649
C03433=1173.149,371.658,-80.330,-176.120,8.857,148.649
C03434=1173.146,371.905,-80.365,-176.118,8.861,148.650
C03435=1173.142,372.153,-80.400,-176.117,8.865,148.650
C03436=1173.137,372.400,-80.436,-176.115,8.868,148.651
C03437=1173.134,372.648,-80.470,-176.113,8.872,148.651
C03438=1173.130,372.895,-80.505,-176.111,8.876,148.652
C03439=1173.126,373.143,-80.540,-176.110,8.880,148.652
C03440=1173.122,373.390,-80.575,-176.109,8.883,148.653
C03441=1173.118,373.638,-80.610,-176.107,8.886,148.653
C03442=1173.114,373.885,-80.645,-176.106,8.890,148.654
C03443=1173.110,374.133,-80.681,-176.104,8.894,148.655
C03444=1173.106,374.380,-80.715,-176.103,8.898,148.655
C03445=1173.102,374.628,-80.751,-176.102,8.901,148.656
C03446=1173.098,374.876,-80.786,-176.100,8.905,148.656
C03447=1173.094,375.123,-80.821,-176.099,8.909,148.657
C03448=1173.090,375.370,-80.856,-176.097,8.912,148.657
C03449=1173.086,375.618,-80.891,-176.096,8.916,148.658
C03450=1173.082,375.865,-80.926,-176.095,8.919,148.658
C03451=1173.078,376.112,-80.962,-176.093,8.923,148.659
C03452=1173.074,376.361,-80.997,-176.092,8.926,148.660
C03453=1173.071,376.608,-81.032,-176.091,8.930,148.660
C03454=1173.066,376.855,-81.068,-176.090,8.933,148.661
C03455=1173.062,377.103,-81.102,-176.089,8.937,148.661
C03456=1173.059,377.350,-81.138,-176.087,8.941,148.662
C03457=1173.054,377.597,-81.173,-176.086,8.944,148.663
C03458=1173.051,377.845,-81.209,-176.085,8.948,148.663
C03459=1173.047,378.093,-81.244,-176.084,8.951,148.664
C03460=1173.043,378.340,-81.279,-176.083,8.955,148.665
C03461=1173.039,378.587,-81.314,-176.082,8.958,148.665
C03462=1173.035,378.835,-81.350,-176.080,8.962,148.666
C03463=1173.031,379.083,-81.386,-176.080,8.965,148.666
C03464=1173.026,379.330,-81.420,-176.078,8.969,148.667
C03465=1173.023,379.577,-81.456,-176.077,8.972,148.667
C03466=1173.019,379.825,-81.491,-176.077,8.975,148.668
C03467=1173.015,380.072,-81.527,-176.075,8.979,148.669
C03468=1173.011,380.319,-81.562,-176.075,8.982,148.669
C03469=1173.007,380.567,-81.597,-176.073,8.986,148.670
C03470=1173.003,380.815,-81.633,-176.072,8.989,148.671
C03471=1172.999,381.062,-81.668,-176.072,8.993,148.671
C03472=1172.995,381.309,-81.704,-176.071,8.996,148.672
C03473=1172.991,381.557,-81.739,-176.070,9.000,148.673
C03474=1172.987,381.804,-81.775,-176.069,9.003,148.673
C03475=1172.984,382.052,-81.811,-176.068,9.006,148.674
C03476=1172.979,382.299,-81.846,-176.068,9.009,148.675
C03477=1172.976,382.546,-81.881,-176.066,9.013,148.675
C03478=1172.972,382.794,-81.917,-176.066,9.017,148.676
C03479=1172.968,383.042,-81.953,-176.065,9.020,148.677
C03480=1172.963,383.289,-81.987,-176.064,9.023,148.677
C03481=1172.960,383.537,-82.023,-176.064,9.026,148.678
C03482=1172.956,383.784,-82.059,-176.063,9.029,148.679
C03483=1172.952,384.032,-82.094,-176.063,9.033,148.679
C03484=1172.948,384.279,-82.130,-176.062,9.036,148.680
C03485=1172.944,384.526,-82.165,-176.061,9.039,148.681
C03486=1172.940,384.774,-82.201,-176.061,9.042,148.681
C03487=1172.936,385.021,-82.237,-176.060,9.046,148.682
C03488=1172.933,385.269,-82.272,-176.059,9.049,148.683
C03489=1172.928,385.516,-82.308,-176.059,9.052,148.683
C03490=1172.924,385.763,-82.343,-176.058,9.056,148.684
C03491=1172.920,386.011,-82.379,-176.058,9.059,148.685
C03492=1172.917,386.258,-82.415,-176.057,9.062,148.685
C03493=1172.912,386.505,-82.451,-176.057,9.065,148.686
C03494=1172.909,386.753,-82.487,-176.056,9.069,148.687
C03495=1172.905,387.000,-82.522,-176.056,9.071,148.688
C03496=1172.901,387.247,-82.558,-176.056,9.075,148.688
C03497=1172.896,387.495,-82.594,-176.055,9.078,148.689
C03498=1172.893,387.743,-82.629,-176.054,9.081,148.690
C03499=1172.889,387.990,-82.665,-176.055,9.084,148.690
C03500=1172.885,388.238,-82.700,-176.054,9.087,148.691
C03501=1172.880,388.485,-82.736,-176.053,9.090,148.692
C03502=1172.877,388.732,-82.772,-176.054,9.093,148.692
C03503=1172.873,388.980,-82.807,-176.053,9.096,148.693
C03504=1172.870,389.227,-82.844,-176.053,9.099,148.694
C03505=1172.865,389.474,-82.880,-176.052,9.102,148.695
C03506=1172.862,389.722,-82.915,-176.053,9.104,148.695
C03507=1172.858,389.969,-82.951,-176.052,9.108,148.696
C03508=1172.853,390.216,-82.987,-176.052,9.110,148.697
C03509=1172.849,390.464,-83.022,-176.052,9.114,148.697
C03510=1172.846,390.711,-83.058,-176.052,9.116,148.698
C03511=1172.842,390.958,-83.094,-176.052,9.120,148.699
C03512=1172.838,391.206,-83.130,-176.051,9.122,148.699
C03513=1172.834,391.491,-83.170,-176.051,9.126,148.700
C03514=1172.829,391.775,-83.212,-176.052,9.128,148.701
C03515=1172.824,392.060,-83.253,-176.051,9.131,148.702
C03516=1172.820,392.345,-83.295,-176.051,9.135,148.703
C03517=1172.816,392.592,-83.331,-176.051,9.138,148.704
C03518=1172.813,392.840,-83.366,-176.051,9.140,148.704
C03519=1172.808,393.088,-83.402,-176.051,9.143,148.705
C03520=1172.805,393.334,-83.439,-176.051,9.146,148.706
C03521=1172.801,393.581,-83.474,-176.051,9.149,148.706
C03522=1172.796,393.829,-83.510,-176.051,9.151,148.707
C03523=1172.792,394.076,-83.545,-176.051,9.154,148.708
C03524=1172.789,394.323,-83.582,-176.051,9.157,148.709
C03525=1172.785,394.571,-83.618,-176.051,9.160,148.709
C03526=1172.781,394.819,-83.653,-176.051,9.162,148.710
C03527=1172.777,395.066,-83.689,-176.051,9.165,148.711
C03528=1172.773,395.313,-83.726,-176.051,9.167,148.711
C03529=1172.770,395.561,-83.761,-176.051,9.170,148.712
C03530=1172.765,395.808,-83.797,-176.051,9.172,148.713
C03531=1172.761,396.055,-83.833,-176.052,9.175,148.713
C03532=1172.758,396.302,-83.869,-176.052,9.177,148.714
C03533=1172.753,396.550,-83.905,-176.052,9.180,148.715
C03534=1172.750,396.798,-83.941,-176.052,9.182,148.716
C03535=1172.746,397.045,-83.976,-176.052,9.185,148.716
C03536=1172.742,397.292,-84.013,-176.052,9.188,148.717
C03537=1172.738,397.540,-84.049,-176.052,9.190,148.718
C03538=1172.734,397.788,-84.085,-176.053,9.193,148.718
C03539=1172.730,398.034,-84.121,-176.052,9.195,148.719
C03540=1172.726,398.281,-84.156,-176.052,9.198,148.720
C03541=1172.722,398.529,-84.192,-176.053,9.199,148.720
C03542=1172.718,398.776,-84.229,-176.053,9.202,148.721
C03543=1172.714,399.024,-84.265,-176.054,9.204,148.722
C03544=1172.710,399.271,-84.300,-176.054,9.207,148.722
C03545=1172.706,399.519,-84.337,-176.054,9.210,148.723
C03546=1172.703,399.766,-84.373,-176.054,9.212,148.724
C03547=1172.699,400.014,-84.408,-176.054,9.214,148.724
C03548=1172.695,400.261,-84.445,-176.054,9.216,148.725
C03549=1172.691,400.508,-84.481,-176.055,9.219,148.726
C03550=1172.687,400.756,-84.517,-176.055,9.221,148.726
C03551=1172.683,401.002,-84.553,-176.055,9.223,148.727
C03552=1172.679,401.250,-84.588,-176.056,9.226,148.728
C03553=1172.675,401.498,-84.624,-176.055,9.228,148.728
C03554=1172.671,401.744,-84.661,-176.056,9.230,148.729
C03555=1172.667,401.992,-84.697,-176.056,9.232,148.730
C03556=1172.663,402.240,-84.732,-176.056,9.235,148.730
C03557=1172.659,402.487,-84.769,-176.057,9.237,148.731
C03558=1172.656,402.734,-84.805,-176.057,9.239,148.732
C03559=1172.652,402.982,-84.840,-176.057,9.241,148.732
C03560=1172.648,403.229,-84.877,-176.058,9.243,148.733
C03561=1172.644,403.477,-84.913,-176.058,9.246,148.734
C03562=1172.640,403.724,-84.949,-176.058,9.248,148.734
C03563=1172.636,403.971,-84.985,-176.058,9.250,148.735
C03564=1172.632,404.219,-85.021,-176.058,9.252,148.736
C03565=1172.629,404.466,-85.057,-176.059,9.254,148.736
C03566=1172.624,404.713,-85.093,-176.059,9.256,148.737
C03567=1172.620,404.960,-85.129,-176.059,9.259,148.737
C03568=1172.616,405.208,-85.166,-176.060,9.260,148.738
C03569=1172.612,405.455,-85.201,-176.059,9.263,148.739
C03570=1172.609,405.702,-85.237,-176.060,9.264,148.739
C03571=1172.604,405.950,-85.274,-176.060,9.267,148.740
C03572=1172.601,406.197,-85.310,-176.061,9.269,148.740
C03573=1172.597,406.445,-85.346,-176.061,9.271,148.741
C03574=1172.593,406.692,-85.382,-176.061,9.273,148.742
C03575=1172.589,406.939,-85.418,-176.061,9.275,148.742
C03576=1172.585,407.187,-85.454,-176.062,9.277,148.743
C03577=1172.581,407.434,-85.491,-176.062,9.279,148.744
C03578=1172.577,407.682,-85.526,-176.062,9.281,148.744
C03579=1172.573,407.929,-85.563,-176.062,9.283,148.745
C03580=1172.570,408.176,-85.599,-176.063,9.285,148.745
C03581=1172.566,408.423,-85.636,-176.063,9.287,148.746
C03582=1172.562,408.671,-85.671,-176.063,9.289,148.746
C03583=1172.558,408.919,-85.707,-176.064,9.291,148.747
C03584=1172.554,409.166,-85.744,-176.064,9.293,148.748
C03585=1172.550,409.413,-85.780,-176.064,9.295,148.748
C03586=1172.546,409.660,-85.816,-176.065,9.297,148.749
C03587=1172.542,409.907,-85.851,-176.065,9.299,148.749
C03588=1172.538,410.154,-85.888,-176.065,9.301,148.750
C03589=1172.534,410.402,-85.924,-176.065,9.303,148.751
C03590=1172.530,410.649,-85.960,-176.066,9.304,148.751
C03591=1172.527,410.896,-85.996,-176.066,9.307,148.752
C03592=1172.523,411.144,-86.033,-176.066,9.308,148.752
C03593=1172.519,411.391,-86.068,-176.067,9.310,148.753
C03594=1172.515,411.638,-86.105,-176.067,9.312,148.754
C03595=1172.511,411.886,-86.141,-176.067,9.314,148.754
C03596=1172.507,412.134,-86.177,-176.067,9.316,148.755
C03597=1172.503,412.381,-86.213,-176.068,9.318,148.755
C03598=1172.499,412.628,-86.249,-176.068,9.319,148.756
C03599=1172.496,412.875,-86.286,-176.068,9.322,148.756
C03600=1172.491,413.123,-86.322,-176.068,9.323,148.757
C03601=1172.487,413.370,-86.359,-176.069,9.325,148.758
C03602=1172.483,413.618,-86.394,-176.069,9.327,148.758
C03603=1172.479,413.865,-86.431,-176.069,9.329,148.759
C03604=1172.476,414.112,-86.467,-176.070,9.330,148.759
C03605=1172.472,414.360,-86.503,-176.069,9.333,148.760
C03606=1172.468,414.607,-86.539,-176.070,9.334,148.760
C03607=1172.464,414.854,-86.576,-176.070,9.336,148.761
C03608=1172.460,415.102,-86.611,-176.070,9.338,148.761
C03609=1172.456,415.349,-86.648,-176.071,9.340,148.762
C03610=1172.453,415.596,-86.684,-176.071,9.341,148.762
C03611=1172.450,415.844,-86.720,-176.071,9.344,148.763
C03612=1172.448,416.091,-86.756,-176.071,9.345,148.763
C03613=1172.449,416.360,-86.795,-176.072,9.347,148.764
C03614=1172.449,416.629,-86.834,-176.072,9.349,148.765
C03615=1172.451,416.897,-86.873,-176.072,9.350,148.765
C03616=1172.454,417.165,-86.911,-176.072,9.352,148.765
C03617=1172.033,417.167,-86.956,-176.075,9.363,148.769
C03618=1172.030,416.895,-86.917,-176.075,9.361,148.769
C03619=1172.028,416.624,-86.877,-176.075,9.360,148.768
C03620=1172.027,416.351,-86.838,-176.075,9.357,148.768
C03621=1172.028,416.080,-86.799,-176.074,9.356,148.767
C03622=1172.029,415.832,-86.762,-176.074,9.355,148.767
C03623=1172.031,415.585,-86.726,-176.074,9.352,148.766
C03624=1172.035,415.338,-86.691,-176.074,9.351,148.766
C03625=1172.039,415.090,-86.654,-176.073,9.349,148.765
C03626=1172.043,414.843,-86.618,-176.073,9.347,148.764
C03627=1172.047,414.596,-86.581,-176.073,9.345,148.764
C03628=1172.050,414.348,-86.546,-176.073,9.344,148.763
C03629=1172.054,414.101,-86.509,-176.073,9.341,148.763
C03630=1172.059,413.853,-86.473,-176.072,9.340,148.762
C03631=1172.062,413.606,-86.437,-176.072,9.338,148.762
C03632=1172.067,413.358,-86.400,-176.072,9.336,148.761
C03633=1172.070,413.112,-86.364,-176.072,9.334,148.761
C03634=1172.074,412.864,-86.328,-176.071,9.332,148.760
C03635=1172.078,412.617,-86.292,-176.071,9.330,148.760
C03636=1172.082,412.369,-86.256,-176.070,9.328,148.759
C03637=1172.085,412.122,-86.219,-176.070,9.327,148.758
C03638=1172.090,411.874,-86.183,-176.070,9.324,148.758
C03639=1172.093,411.627,-86.147,-176.070,9.323,148.757
C03640=1172.098,411.380,-86.111,-176.069,9.322,148.757
C03641=1172.102,411.134,-86.075,-176.069,9.319,148.756
C03642=1172.106,410.886,-86.039,-176.069,9.318,148.756
C03643=1172.109,410.639,-86.002,-176.068,9.316,148.755
C03644=1172.114,410.391,-85.966,-176.069,9.314,148.754
C03645=1172.117,410.144,-85.930,-176.068,9.312,148.754
C03646=1172.122,409.896,-85.894,-176.068,9.309,148.753
C03647=1172.125,409.649,-85.858,-176.067,9.308,148.753
C03648=1172.129,409.402,-85.822,-176.067,9.306,148.752
C03649=1172.133,409.155,-85.785,-176.067,9.304,148.751
C03650=1172.137,408.907,-85.749,-176.066,9.302,148.751
C03651=1172.141,408.659,-85.714,-176.067,9.300,148.750
C03652=1172.145,408.412,-85.677,-176.066,9.298,148.750
C03653=1172.148,408.165,-85.641,-176.066,9.296,148.749
C03654=1172.153,407.918,-85.604,-176.065,9.294,148.748
C03655=1172.156,407.670,-85.569,-176.065,9.292,148.748
C03656=1172.160,407.423,-85.532,-176.065,9.290,148.747
C03657=1172.164,407.175,-85.496,-176.064,9.288,148.747
C03658=1172.168,406.928,-85.460,-176.064,9.286,148.746
